        IF finalPosition == 13 THEN
          ;FOLD SPTP P113 Vel=100 % PDAT1 Tool[1]:SMC Base[0] ;%{PE}
          ;FOLD Parameters ;%{h}
          ;Params IlfProvider=kukaroboter.basistech.inlineforms.movement.spline; Kuka.IsGlobalPoint=False; Kuka.PointName=P113; Kuka.BlendingEnabled=False; Kuka.MoveDataPtpName=PDAT1; Kuka.VelocityPtp=100; Kuka.VelocityFieldEnabled=True; Kuka.ColDetectFieldEnabled=True; Kuka.CurrentCDSetIndex=0; Kuka.MovementParameterFieldEnabled=True; IlfCommand=SPTP
          ;ENDFOLD
          SPTP XP113 WITH $VEL_AXIS[1] = SVEL_JOINT(100.0), $TOOL = STOOL2(FP113), $BASE = SBASE(FP113.BASE_NO), $IPO_MODE = SIPO_MODE(FP113.IPO_FRAME), $LOAD = SLOAD(FP113.TOOL_NO), $ACC_AXIS[1] = SACC_JOINT(PPDAT1), $APO = SAPO_PTP(PPDAT1), $GEAR_JERK[1] = SGEAR_JERK(PPDAT1), $COLLMON_TOL_PRO[1] = USE_CM_PRO_VALUES(0)
          ;ENDFOLD
          ;FOLD SLIN P213 Vel=0.1 m/s CPDAT27 Tool[1]:SMC Base[0] ;%{PE}
          ;FOLD Parameters ;%{h}
          ;Params IlfProvider=kukaroboter.basistech.inlineforms.movement.spline; Kuka.IsGlobalPoint=False; Kuka.PointName=P213; Kuka.BlendingEnabled=False; Kuka.MoveDataName=CPDAT27; Kuka.VelocityPath=0.1; Kuka.VelocityFieldEnabled=True; Kuka.ColDetectFieldEnabled=True; Kuka.CurrentCDSetIndex=0; Kuka.MovementParameterFieldEnabled=True; IlfCommand=SLIN
          ;ENDFOLD
          SLIN XP213 WITH $VEL = SVEL_CP(0.1, , LCPDAT27), $TOOL = STOOL2(FP213), $BASE = SBASE(FP213.BASE_NO), $IPO_MODE = SIPO_MODE(FP213.IPO_FRAME), $LOAD = SLOAD(FP213.TOOL_NO), $ACC = SACC_CP(LCPDAT27), $ORI_TYPE = SORI_TYP(LCPDAT27), $APO = SAPO(LCPDAT27), $JERK = SJERK(LCPDAT27), $COLLMON_TOL_PRO[1] = USE_CM_PRO_VALUES(0)
          ;ENDFOLD
          ;FOLD Gripper SET [1]Gripper1 State=[1]ABIERTA Wait 0.2[s] Check with Strategy 1 ;%{PE}
          ;FOLD Parameters Parameters ;%{h}
          ;Params IlfProvider=GripperTech.GripperSet;setgripper=1;setstate=1;setcont=nocont;waittime=0.2;errorstrategy=1
          ;ENDFOLD
          GRPg_SetStateAndCheck(1, 1, 0.2, 1)
          ;ENDFOLD
          ;FOLD SLIN P113 Vel=0.1 m/s CPDAT28 Tool[1]:SMC Base[0] ;%{PE}
          ;FOLD Parameters ;%{h}
          ;Params IlfProvider=kukaroboter.basistech.inlineforms.movement.spline; Kuka.IsGlobalPoint=False; Kuka.PointName=P113; Kuka.BlendingEnabled=False; Kuka.MoveDataName=CPDAT28; Kuka.VelocityPath=0.1; Kuka.VelocityFieldEnabled=True; Kuka.ColDetectFieldEnabled=True; Kuka.CurrentCDSetIndex=0; Kuka.MovementParameterFieldEnabled=True; IlfCommand=SLIN
          ;ENDFOLD
          SLIN XP113 WITH $VEL = SVEL_CP(0.1, , LCPDAT28), $TOOL = STOOL2(FP113), $BASE = SBASE(FP113.BASE_NO), $IPO_MODE = SIPO_MODE(FP113.IPO_FRAME), $LOAD = SLOAD(FP113.TOOL_NO), $ACC = SACC_CP(LCPDAT28), $ORI_TYPE = SORI_TYP(LCPDAT28), $APO = SAPO(LCPDAT28), $JERK = SJERK(LCPDAT28), $COLLMON_TOL_PRO[1] = USE_CM_PRO_VALUES(0)
          ;ENDFOLD
          ;FOLD SPTP P600 Vel=100 % PDAT1 Tool[1]:SMC Base[0] ;%{PE}
          ;FOLD Parameters ;%{h}
          ;Params IlfProvider=kukaroboter.basistech.inlineforms.movement.spline; Kuka.IsGlobalPoint=False; Kuka.PointName=P600; Kuka.BlendingEnabled=False; Kuka.MoveDataPtpName=PDAT1; Kuka.VelocityPtp=100; Kuka.VelocityFieldEnabled=True; Kuka.ColDetectFieldEnabled=True; Kuka.CurrentCDSetIndex=0; Kuka.MovementParameterFieldEnabled=True; IlfCommand=SPTP
          ;ENDFOLD
          SPTP XP600 WITH $VEL_AXIS[1] = SVEL_JOINT(100.0), $TOOL = STOOL2(FP600), $BASE = SBASE(FP600.BASE_NO), $IPO_MODE = SIPO_MODE(FP600.IPO_FRAME), $LOAD = SLOAD(FP600.TOOL_NO), $ACC_AXIS[1] = SACC_JOINT(PPDAT1), $APO = SAPO_PTP(PPDAT1), $GEAR_JERK[1] = SGEAR_JERK(PPDAT1), $COLLMON_TOL_PRO[1] = USE_CM_PRO_VALUES(0)
          ;ENDFOLD
          ;FOLD SLIN P601 Vel=0.1 m/s CPDAT27 Tool[1]:SMC Base[0] ;%{PE}
          ;FOLD Parameters ;%{h}
          ;Params IlfProvider=kukaroboter.basistech.inlineforms.movement.spline; Kuka.IsGlobalPoint=False; Kuka.PointName=P601; Kuka.BlendingEnabled=False; Kuka.MoveDataName=CPDAT27; Kuka.VelocityPath=0.1; Kuka.VelocityFieldEnabled=True; Kuka.ColDetectFieldEnabled=True; Kuka.CurrentCDSetIndex=0; Kuka.MovementParameterFieldEnabled=True; IlfCommand=SLIN
          ;ENDFOLD
          SLIN XP601 WITH $VEL = SVEL_CP(0.1, , LCPDAT27), $TOOL = STOOL2(FP601), $BASE = SBASE(FP601.BASE_NO), $IPO_MODE = SIPO_MODE(FP601.IPO_FRAME), $LOAD = SLOAD(FP601.TOOL_NO), $ACC = SACC_CP(LCPDAT27), $ORI_TYPE = SORI_TYP(LCPDAT27), $APO = SAPO(LCPDAT27), $JERK = SJERK(LCPDAT27), $COLLMON_TOL_PRO[1] = USE_CM_PRO_VALUES(0)
          ;ENDFOLD
          ;FOLD SLIN P602 Vel=0.1 m/s CPDAT27 Tool[1]:SMC Base[0] ;%{PE}
          ;FOLD Parameters ;%{h}
          ;Params IlfProvider=kukaroboter.basistech.inlineforms.movement.spline; Kuka.IsGlobalPoint=False; Kuka.PointName=P602; Kuka.BlendingEnabled=False; Kuka.MoveDataName=CPDAT27; Kuka.VelocityPath=0.1; Kuka.VelocityFieldEnabled=True; Kuka.ColDetectFieldEnabled=True; Kuka.CurrentCDSetIndex=0; Kuka.MovementParameterFieldEnabled=True; IlfCommand=SLIN
          ;ENDFOLD
          SLIN XP602 WITH $VEL = SVEL_CP(0.1, , LCPDAT27), $TOOL = STOOL2(FP602), $BASE = SBASE(FP602.BASE_NO), $IPO_MODE = SIPO_MODE(FP602.IPO_FRAME), $LOAD = SLOAD(FP602.TOOL_NO), $ACC = SACC_CP(LCPDAT27), $ORI_TYPE = SORI_TYP(LCPDAT27), $APO = SAPO(LCPDAT27), $JERK = SJERK(LCPDAT27), $COLLMON_TOL_PRO[1] = USE_CM_PRO_VALUES(0)
          ;ENDFOLD
        ENDIF
        IF finalPosition == 14 THEN
          ;FOLD SPTP P114 Vel=100 % PDAT1 Tool[1]:SMC Base[0] ;%{PE}
          ;FOLD Parameters ;%{h}
          ;Params IlfProvider=kukaroboter.basistech.inlineforms.movement.spline; Kuka.IsGlobalPoint=False; Kuka.PointName=P114; Kuka.BlendingEnabled=False; Kuka.MoveDataPtpName=PDAT1; Kuka.VelocityPtp=100; Kuka.VelocityFieldEnabled=True; Kuka.ColDetectFieldEnabled=True; Kuka.CurrentCDSetIndex=0; Kuka.MovementParameterFieldEnabled=True; IlfCommand=SPTP
          ;ENDFOLD
          SPTP XP114 WITH $VEL_AXIS[1] = SVEL_JOINT(100.0), $TOOL = STOOL2(FP114), $BASE = SBASE(FP114.BASE_NO), $IPO_MODE = SIPO_MODE(FP114.IPO_FRAME), $LOAD = SLOAD(FP114.TOOL_NO), $ACC_AXIS[1] = SACC_JOINT(PPDAT1), $APO = SAPO_PTP(PPDAT1), $GEAR_JERK[1] = SGEAR_JERK(PPDAT1), $COLLMON_TOL_PRO[1] = USE_CM_PRO_VALUES(0)
          ;ENDFOLD
          ;FOLD SLIN P214 Vel=0.1 m/s CPDAT27 Tool[1]:SMC Base[0] ;%{PE}
          ;FOLD Parameters ;%{h}
          ;Params IlfProvider=kukaroboter.basistech.inlineforms.movement.spline; Kuka.IsGlobalPoint=False; Kuka.PointName=P214; Kuka.BlendingEnabled=False; Kuka.MoveDataName=CPDAT27; Kuka.VelocityPath=0.1; Kuka.VelocityFieldEnabled=True; Kuka.ColDetectFieldEnabled=True; Kuka.CurrentCDSetIndex=0; Kuka.MovementParameterFieldEnabled=True; IlfCommand=SLIN
          ;ENDFOLD
          SLIN XP214 WITH $VEL = SVEL_CP(0.1, , LCPDAT27), $TOOL = STOOL2(FP214), $BASE = SBASE(FP214.BASE_NO), $IPO_MODE = SIPO_MODE(FP214.IPO_FRAME), $LOAD = SLOAD(FP214.TOOL_NO), $ACC = SACC_CP(LCPDAT27), $ORI_TYPE = SORI_TYP(LCPDAT27), $APO = SAPO(LCPDAT27), $JERK = SJERK(LCPDAT27), $COLLMON_TOL_PRO[1] = USE_CM_PRO_VALUES(0)
          ;ENDFOLD
          ;FOLD Gripper SET [1]Gripper1 State=[1]ABIERTA Wait 0.2[s] Check with Strategy 1 ;%{PE}
          ;FOLD Parameters Parameters ;%{h}
          ;Params IlfProvider=GripperTech.GripperSet;setgripper=1;setstate=1;setcont=nocont;waittime=0.2;errorstrategy=1
          ;ENDFOLD
          GRPg_SetStateAndCheck(1, 1, 0.2, 1)
          ;ENDFOLD
          ;FOLD SLIN P114 Vel=0.1 m/s CPDAT28 Tool[1]:SMC Base[0] ;%{PE}
          ;FOLD Parameters ;%{h}
          ;Params IlfProvider=kukaroboter.basistech.inlineforms.movement.spline; Kuka.IsGlobalPoint=False; Kuka.PointName=P114; Kuka.BlendingEnabled=False; Kuka.MoveDataName=CPDAT28; Kuka.VelocityPath=0.1; Kuka.VelocityFieldEnabled=True; Kuka.ColDetectFieldEnabled=True; Kuka.CurrentCDSetIndex=0; Kuka.MovementParameterFieldEnabled=True; IlfCommand=SLIN
          ;ENDFOLD
          SLIN XP114 WITH $VEL = SVEL_CP(0.1, , LCPDAT28), $TOOL = STOOL2(FP114), $BASE = SBASE(FP114.BASE_NO), $IPO_MODE = SIPO_MODE(FP114.IPO_FRAME), $LOAD = SLOAD(FP114.TOOL_NO), $ACC = SACC_CP(LCPDAT28), $ORI_TYPE = SORI_TYP(LCPDAT28), $APO = SAPO(LCPDAT28), $JERK = SJERK(LCPDAT28), $COLLMON_TOL_PRO[1] = USE_CM_PRO_VALUES(0)
          ;ENDFOLD
          ;FOLD SPTP P600 Vel=100 % PDAT1 Tool[1]:SMC Base[0] ;%{PE}
          ;FOLD Parameters ;%{h}
          ;Params IlfProvider=kukaroboter.basistech.inlineforms.movement.spline; Kuka.IsGlobalPoint=False; Kuka.PointName=P600; Kuka.BlendingEnabled=False; Kuka.MoveDataPtpName=PDAT1; Kuka.VelocityPtp=100; Kuka.VelocityFieldEnabled=True; Kuka.ColDetectFieldEnabled=True; Kuka.CurrentCDSetIndex=0; Kuka.MovementParameterFieldEnabled=True; IlfCommand=SPTP
          ;ENDFOLD
          SPTP XP600 WITH $VEL_AXIS[1] = SVEL_JOINT(100.0), $TOOL = STOOL2(FP600), $BASE = SBASE(FP600.BASE_NO), $IPO_MODE = SIPO_MODE(FP600.IPO_FRAME), $LOAD = SLOAD(FP600.TOOL_NO), $ACC_AXIS[1] = SACC_JOINT(PPDAT1), $APO = SAPO_PTP(PPDAT1), $GEAR_JERK[1] = SGEAR_JERK(PPDAT1), $COLLMON_TOL_PRO[1] = USE_CM_PRO_VALUES(0)
          ;ENDFOLD
          ;FOLD SLIN P601 Vel=0.1 m/s CPDAT27 Tool[1]:SMC Base[0] ;%{PE}
          ;FOLD Parameters ;%{h}
          ;Params IlfProvider=kukaroboter.basistech.inlineforms.movement.spline; Kuka.IsGlobalPoint=False; Kuka.PointName=P601; Kuka.BlendingEnabled=False; Kuka.MoveDataName=CPDAT27; Kuka.VelocityPath=0.1; Kuka.VelocityFieldEnabled=True; Kuka.ColDetectFieldEnabled=True; Kuka.CurrentCDSetIndex=0; Kuka.MovementParameterFieldEnabled=True; IlfCommand=SLIN
          ;ENDFOLD
          SLIN XP601 WITH $VEL = SVEL_CP(0.1, , LCPDAT27), $TOOL = STOOL2(FP601), $BASE = SBASE(FP601.BASE_NO), $IPO_MODE = SIPO_MODE(FP601.IPO_FRAME), $LOAD = SLOAD(FP601.TOOL_NO), $ACC = SACC_CP(LCPDAT27), $ORI_TYPE = SORI_TYP(LCPDAT27), $APO = SAPO(LCPDAT27), $JERK = SJERK(LCPDAT27), $COLLMON_TOL_PRO[1] = USE_CM_PRO_VALUES(0)
          ;ENDFOLD
          ;FOLD SLIN P602 Vel=0.1 m/s CPDAT27 Tool[1]:SMC Base[0] ;%{PE}
          ;FOLD Parameters ;%{h}
          ;Params IlfProvider=kukaroboter.basistech.inlineforms.movement.spline; Kuka.IsGlobalPoint=False; Kuka.PointName=P602; Kuka.BlendingEnabled=False; Kuka.MoveDataName=CPDAT27; Kuka.VelocityPath=0.1; Kuka.VelocityFieldEnabled=True; Kuka.ColDetectFieldEnabled=True; Kuka.CurrentCDSetIndex=0; Kuka.MovementParameterFieldEnabled=True; IlfCommand=SLIN
          ;ENDFOLD
          SLIN XP602 WITH $VEL = SVEL_CP(0.1, , LCPDAT27), $TOOL = STOOL2(FP602), $BASE = SBASE(FP602.BASE_NO), $IPO_MODE = SIPO_MODE(FP602.IPO_FRAME), $LOAD = SLOAD(FP602.TOOL_NO), $ACC = SACC_CP(LCPDAT27), $ORI_TYPE = SORI_TYP(LCPDAT27), $APO = SAPO(LCPDAT27), $JERK = SJERK(LCPDAT27), $COLLMON_TOL_PRO[1] = USE_CM_PRO_VALUES(0)
          ;ENDFOLD
        ENDIF
        IF finalPosition == 15 THEN
          ;FOLD SPTP P115 Vel=100 % PDAT1 Tool[1]:SMC Base[0] ;%{PE}
          ;FOLD Parameters ;%{h}
          ;Params IlfProvider=kukaroboter.basistech.inlineforms.movement.spline; Kuka.IsGlobalPoint=False; Kuka.PointName=P115; Kuka.BlendingEnabled=False; Kuka.MoveDataPtpName=PDAT1; Kuka.VelocityPtp=100; Kuka.VelocityFieldEnabled=True; Kuka.ColDetectFieldEnabled=True; Kuka.CurrentCDSetIndex=0; Kuka.MovementParameterFieldEnabled=True; IlfCommand=SPTP
          ;ENDFOLD
          SPTP XP115 WITH $VEL_AXIS[1] = SVEL_JOINT(100.0), $TOOL = STOOL2(FP115), $BASE = SBASE(FP115.BASE_NO), $IPO_MODE = SIPO_MODE(FP115.IPO_FRAME), $LOAD = SLOAD(FP115.TOOL_NO), $ACC_AXIS[1] = SACC_JOINT(PPDAT1), $APO = SAPO_PTP(PPDAT1), $GEAR_JERK[1] = SGEAR_JERK(PPDAT1), $COLLMON_TOL_PRO[1] = USE_CM_PRO_VALUES(0)
          ;ENDFOLD
          ;FOLD SLIN P215 Vel=0.1 m/s CPDAT27 Tool[1]:SMC Base[0] ;%{PE}
          ;FOLD Parameters ;%{h}
          ;Params IlfProvider=kukaroboter.basistech.inlineforms.movement.spline; Kuka.IsGlobalPoint=False; Kuka.PointName=P215; Kuka.BlendingEnabled=False; Kuka.MoveDataName=CPDAT27; Kuka.VelocityPath=0.1; Kuka.VelocityFieldEnabled=True; Kuka.ColDetectFieldEnabled=True; Kuka.CurrentCDSetIndex=0; Kuka.MovementParameterFieldEnabled=True; IlfCommand=SLIN
          ;ENDFOLD
          SLIN XP215 WITH $VEL = SVEL_CP(0.1, , LCPDAT27), $TOOL = STOOL2(FP215), $BASE = SBASE(FP215.BASE_NO), $IPO_MODE = SIPO_MODE(FP215.IPO_FRAME), $LOAD = SLOAD(FP215.TOOL_NO), $ACC = SACC_CP(LCPDAT27), $ORI_TYPE = SORI_TYP(LCPDAT27), $APO = SAPO(LCPDAT27), $JERK = SJERK(LCPDAT27), $COLLMON_TOL_PRO[1] = USE_CM_PRO_VALUES(0)
          ;ENDFOLD
          ;FOLD Gripper SET [1]Gripper1 State=[1]ABIERTA Wait 0.2[s] Check with Strategy 1 ;%{PE}
          ;FOLD Parameters Parameters ;%{h}
          ;Params IlfProvider=GripperTech.GripperSet;setgripper=1;setstate=1;setcont=nocont;waittime=0.2;errorstrategy=1
          ;ENDFOLD
          GRPg_SetStateAndCheck(1, 1, 0.2, 1)
          ;ENDFOLD
          ;FOLD SLIN P115 Vel=0.1 m/s CPDAT28 Tool[1]:SMC Base[0] ;%{PE}
          ;FOLD Parameters ;%{h}
          ;Params IlfProvider=kukaroboter.basistech.inlineforms.movement.spline; Kuka.IsGlobalPoint=False; Kuka.PointName=P115; Kuka.BlendingEnabled=False; Kuka.MoveDataName=CPDAT28; Kuka.VelocityPath=0.1; Kuka.VelocityFieldEnabled=True; Kuka.ColDetectFieldEnabled=True; Kuka.CurrentCDSetIndex=0; Kuka.MovementParameterFieldEnabled=True; IlfCommand=SLIN
          ;ENDFOLD
          SLIN XP115 WITH $VEL = SVEL_CP(0.1, , LCPDAT28), $TOOL = STOOL2(FP115), $BASE = SBASE(FP115.BASE_NO), $IPO_MODE = SIPO_MODE(FP115.IPO_FRAME), $LOAD = SLOAD(FP115.TOOL_NO), $ACC = SACC_CP(LCPDAT28), $ORI_TYPE = SORI_TYP(LCPDAT28), $APO = SAPO(LCPDAT28), $JERK = SJERK(LCPDAT28), $COLLMON_TOL_PRO[1] = USE_CM_PRO_VALUES(0)
          ;ENDFOLD
          ;FOLD SPTP P600 Vel=100 % PDAT1 Tool[1]:SMC Base[0] ;%{PE}
          ;FOLD Parameters ;%{h}
          ;Params IlfProvider=kukaroboter.basistech.inlineforms.movement.spline; Kuka.IsGlobalPoint=False; Kuka.PointName=P600; Kuka.BlendingEnabled=False; Kuka.MoveDataPtpName=PDAT1; Kuka.VelocityPtp=100; Kuka.VelocityFieldEnabled=True; Kuka.ColDetectFieldEnabled=True; Kuka.CurrentCDSetIndex=0; Kuka.MovementParameterFieldEnabled=True; IlfCommand=SPTP
          ;ENDFOLD
          SPTP XP600 WITH $VEL_AXIS[1] = SVEL_JOINT(100.0), $TOOL = STOOL2(FP600), $BASE = SBASE(FP600.BASE_NO), $IPO_MODE = SIPO_MODE(FP600.IPO_FRAME), $LOAD = SLOAD(FP600.TOOL_NO), $ACC_AXIS[1] = SACC_JOINT(PPDAT1), $APO = SAPO_PTP(PPDAT1), $GEAR_JERK[1] = SGEAR_JERK(PPDAT1), $COLLMON_TOL_PRO[1] = USE_CM_PRO_VALUES(0)
          ;ENDFOLD
          ;FOLD SLIN P601 Vel=0.1 m/s CPDAT27 Tool[1]:SMC Base[0] ;%{PE}
          ;FOLD Parameters ;%{h}
          ;Params IlfProvider=kukaroboter.basistech.inlineforms.movement.spline; Kuka.IsGlobalPoint=False; Kuka.PointName=P601; Kuka.BlendingEnabled=False; Kuka.MoveDataName=CPDAT27; Kuka.VelocityPath=0.1; Kuka.VelocityFieldEnabled=True; Kuka.ColDetectFieldEnabled=True; Kuka.CurrentCDSetIndex=0; Kuka.MovementParameterFieldEnabled=True; IlfCommand=SLIN
          ;ENDFOLD
          SLIN XP601 WITH $VEL = SVEL_CP(0.1, , LCPDAT27), $TOOL = STOOL2(FP601), $BASE = SBASE(FP601.BASE_NO), $IPO_MODE = SIPO_MODE(FP601.IPO_FRAME), $LOAD = SLOAD(FP601.TOOL_NO), $ACC = SACC_CP(LCPDAT27), $ORI_TYPE = SORI_TYP(LCPDAT27), $APO = SAPO(LCPDAT27), $JERK = SJERK(LCPDAT27), $COLLMON_TOL_PRO[1] = USE_CM_PRO_VALUES(0)
          ;ENDFOLD
          ;FOLD SLIN P602 Vel=0.1 m/s CPDAT27 Tool[1]:SMC Base[0] ;%{PE}
          ;FOLD Parameters ;%{h}
          ;Params IlfProvider=kukaroboter.basistech.inlineforms.movement.spline; Kuka.IsGlobalPoint=False; Kuka.PointName=P602; Kuka.BlendingEnabled=False; Kuka.MoveDataName=CPDAT27; Kuka.VelocityPath=0.1; Kuka.VelocityFieldEnabled=True; Kuka.ColDetectFieldEnabled=True; Kuka.CurrentCDSetIndex=0; Kuka.MovementParameterFieldEnabled=True; IlfCommand=SLIN
          ;ENDFOLD
          SLIN XP602 WITH $VEL = SVEL_CP(0.1, , LCPDAT27), $TOOL = STOOL2(FP602), $BASE = SBASE(FP602.BASE_NO), $IPO_MODE = SIPO_MODE(FP602.IPO_FRAME), $LOAD = SLOAD(FP602.TOOL_NO), $ACC = SACC_CP(LCPDAT27), $ORI_TYPE = SORI_TYP(LCPDAT27), $APO = SAPO(LCPDAT27), $JERK = SJERK(LCPDAT27), $COLLMON_TOL_PRO[1] = USE_CM_PRO_VALUES(0)
          ;ENDFOLD
        ENDIF
        IF finalPosition == 16 THEN
          ;FOLD SPTP P116 Vel=100 % PDAT1 Tool[1]:SMC Base[0] ;%{PE}
          ;FOLD Parameters ;%{h}
          ;Params IlfProvider=kukaroboter.basistech.inlineforms.movement.spline; Kuka.IsGlobalPoint=False; Kuka.PointName=P116; Kuka.BlendingEnabled=False; Kuka.MoveDataPtpName=PDAT1; Kuka.VelocityPtp=100; Kuka.VelocityFieldEnabled=True; Kuka.ColDetectFieldEnabled=True; Kuka.CurrentCDSetIndex=0; Kuka.MovementParameterFieldEnabled=True; IlfCommand=SPTP
          ;ENDFOLD
          SPTP XP116 WITH $VEL_AXIS[1] = SVEL_JOINT(100.0), $TOOL = STOOL2(FP116), $BASE = SBASE(FP116.BASE_NO), $IPO_MODE = SIPO_MODE(FP116.IPO_FRAME), $LOAD = SLOAD(FP116.TOOL_NO), $ACC_AXIS[1] = SACC_JOINT(PPDAT1), $APO = SAPO_PTP(PPDAT1), $GEAR_JERK[1] = SGEAR_JERK(PPDAT1), $COLLMON_TOL_PRO[1] = USE_CM_PRO_VALUES(0)
          ;ENDFOLD
          ;FOLD SLIN P216 Vel=0.1 m/s CPDAT27 Tool[1]:SMC Base[0] ;%{PE}
          ;FOLD Parameters ;%{h}
          ;Params IlfProvider=kukaroboter.basistech.inlineforms.movement.spline; Kuka.IsGlobalPoint=False; Kuka.PointName=P216; Kuka.BlendingEnabled=False; Kuka.MoveDataName=CPDAT27; Kuka.VelocityPath=0.1; Kuka.VelocityFieldEnabled=True; Kuka.ColDetectFieldEnabled=True; Kuka.CurrentCDSetIndex=0; Kuka.MovementParameterFieldEnabled=True; IlfCommand=SLIN
          ;ENDFOLD
          SLIN XP216 WITH $VEL = SVEL_CP(0.1, , LCPDAT27), $TOOL = STOOL2(FP216), $BASE = SBASE(FP216.BASE_NO), $IPO_MODE = SIPO_MODE(FP216.IPO_FRAME), $LOAD = SLOAD(FP216.TOOL_NO), $ACC = SACC_CP(LCPDAT27), $ORI_TYPE = SORI_TYP(LCPDAT27), $APO = SAPO(LCPDAT27), $JERK = SJERK(LCPDAT27), $COLLMON_TOL_PRO[1] = USE_CM_PRO_VALUES(0)
          ;ENDFOLD
          ;FOLD Gripper SET [1]Gripper1 State=[1]ABIERTA Wait 0.2[s] Check with Strategy 1 ;%{PE}
          ;FOLD Parameters Parameters ;%{h}
          ;Params IlfProvider=GripperTech.GripperSet;setgripper=1;setstate=1;setcont=nocont;waittime=0.2;errorstrategy=1
          ;ENDFOLD
          GRPg_SetStateAndCheck(1, 1, 0.2, 1)
          ;ENDFOLD
          ;FOLD SLIN P116 Vel=0.1 m/s CPDAT28 Tool[1]:SMC Base[0] ;%{PE}
          ;FOLD Parameters ;%{h}
          ;Params IlfProvider=kukaroboter.basistech.inlineforms.movement.spline; Kuka.IsGlobalPoint=False; Kuka.PointName=P116; Kuka.BlendingEnabled=False; Kuka.MoveDataName=CPDAT28; Kuka.VelocityPath=0.1; Kuka.VelocityFieldEnabled=True; Kuka.ColDetectFieldEnabled=True; Kuka.CurrentCDSetIndex=0; Kuka.MovementParameterFieldEnabled=True; IlfCommand=SLIN
          ;ENDFOLD
          SLIN XP116 WITH $VEL = SVEL_CP(0.1, , LCPDAT28), $TOOL = STOOL2(FP116), $BASE = SBASE(FP116.BASE_NO), $IPO_MODE = SIPO_MODE(FP116.IPO_FRAME), $LOAD = SLOAD(FP116.TOOL_NO), $ACC = SACC_CP(LCPDAT28), $ORI_TYPE = SORI_TYP(LCPDAT28), $APO = SAPO(LCPDAT28), $JERK = SJERK(LCPDAT28), $COLLMON_TOL_PRO[1] = USE_CM_PRO_VALUES(0)
          ;ENDFOLD
          ;FOLD SPTP P600 Vel=100 % PDAT1 Tool[1]:SMC Base[0] ;%{PE}
          ;FOLD Parameters ;%{h}
          ;Params IlfProvider=kukaroboter.basistech.inlineforms.movement.spline; Kuka.IsGlobalPoint=False; Kuka.PointName=P600; Kuka.BlendingEnabled=False; Kuka.MoveDataPtpName=PDAT1; Kuka.VelocityPtp=100; Kuka.VelocityFieldEnabled=True; Kuka.ColDetectFieldEnabled=True; Kuka.CurrentCDSetIndex=0; Kuka.MovementParameterFieldEnabled=True; IlfCommand=SPTP
          ;ENDFOLD
          SPTP XP600 WITH $VEL_AXIS[1] = SVEL_JOINT(100.0), $TOOL = STOOL2(FP600), $BASE = SBASE(FP600.BASE_NO), $IPO_MODE = SIPO_MODE(FP600.IPO_FRAME), $LOAD = SLOAD(FP600.TOOL_NO), $ACC_AXIS[1] = SACC_JOINT(PPDAT1), $APO = SAPO_PTP(PPDAT1), $GEAR_JERK[1] = SGEAR_JERK(PPDAT1), $COLLMON_TOL_PRO[1] = USE_CM_PRO_VALUES(0)
          ;ENDFOLD
          ;FOLD SLIN P601 Vel=0.1 m/s CPDAT27 Tool[1]:SMC Base[0] ;%{PE}
          ;FOLD Parameters ;%{h}
          ;Params IlfProvider=kukaroboter.basistech.inlineforms.movement.spline; Kuka.IsGlobalPoint=False; Kuka.PointName=P601; Kuka.BlendingEnabled=False; Kuka.MoveDataName=CPDAT27; Kuka.VelocityPath=0.1; Kuka.VelocityFieldEnabled=True; Kuka.ColDetectFieldEnabled=True; Kuka.CurrentCDSetIndex=0; Kuka.MovementParameterFieldEnabled=True; IlfCommand=SLIN
          ;ENDFOLD
          SLIN XP601 WITH $VEL = SVEL_CP(0.1, , LCPDAT27), $TOOL = STOOL2(FP601), $BASE = SBASE(FP601.BASE_NO), $IPO_MODE = SIPO_MODE(FP601.IPO_FRAME), $LOAD = SLOAD(FP601.TOOL_NO), $ACC = SACC_CP(LCPDAT27), $ORI_TYPE = SORI_TYP(LCPDAT27), $APO = SAPO(LCPDAT27), $JERK = SJERK(LCPDAT27), $COLLMON_TOL_PRO[1] = USE_CM_PRO_VALUES(0)
          ;ENDFOLD
          ;FOLD SLIN P602 Vel=0.1 m/s CPDAT27 Tool[1]:SMC Base[0] ;%{PE}
          ;FOLD Parameters ;%{h}
          ;Params IlfProvider=kukaroboter.basistech.inlineforms.movement.spline; Kuka.IsGlobalPoint=False; Kuka.PointName=P602; Kuka.BlendingEnabled=False; Kuka.MoveDataName=CPDAT27; Kuka.VelocityPath=0.1; Kuka.VelocityFieldEnabled=True; Kuka.ColDetectFieldEnabled=True; Kuka.CurrentCDSetIndex=0; Kuka.MovementParameterFieldEnabled=True; IlfCommand=SLIN
          ;ENDFOLD
          SLIN XP602 WITH $VEL = SVEL_CP(0.1, , LCPDAT27), $TOOL = STOOL2(FP602), $BASE = SBASE(FP602.BASE_NO), $IPO_MODE = SIPO_MODE(FP602.IPO_FRAME), $LOAD = SLOAD(FP602.TOOL_NO), $ACC = SACC_CP(LCPDAT27), $ORI_TYPE = SORI_TYP(LCPDAT27), $APO = SAPO(LCPDAT27), $JERK = SJERK(LCPDAT27), $COLLMON_TOL_PRO[1] = USE_CM_PRO_VALUES(0)
          ;ENDFOLD
        ENDIF
        IF finalPosition == 17 THEN
          ;FOLD SPTP P117 Vel=100 % PDAT1 Tool[1]:SMC Base[0] ;%{PE}
          ;FOLD Parameters ;%{h}
          ;Params IlfProvider=kukaroboter.basistech.inlineforms.movement.spline; Kuka.IsGlobalPoint=False; Kuka.PointName=P117; Kuka.BlendingEnabled=False; Kuka.MoveDataPtpName=PDAT1; Kuka.VelocityPtp=100; Kuka.VelocityFieldEnabled=True; Kuka.ColDetectFieldEnabled=True; Kuka.CurrentCDSetIndex=0; Kuka.MovementParameterFieldEnabled=True; IlfCommand=SPTP
          ;ENDFOLD
          SPTP XP117 WITH $VEL_AXIS[1] = SVEL_JOINT(100.0), $TOOL = STOOL2(FP117), $BASE = SBASE(FP117.BASE_NO), $IPO_MODE = SIPO_MODE(FP117.IPO_FRAME), $LOAD = SLOAD(FP117.TOOL_NO), $ACC_AXIS[1] = SACC_JOINT(PPDAT1), $APO = SAPO_PTP(PPDAT1), $GEAR_JERK[1] = SGEAR_JERK(PPDAT1), $COLLMON_TOL_PRO[1] = USE_CM_PRO_VALUES(0)
          ;ENDFOLD
          ;FOLD SLIN P217 Vel=0.1 m/s CPDAT27 Tool[1]:SMC Base[0] ;%{PE}
          ;FOLD Parameters ;%{h}
          ;Params IlfProvider=kukaroboter.basistech.inlineforms.movement.spline; Kuka.IsGlobalPoint=False; Kuka.PointName=P217; Kuka.BlendingEnabled=False; Kuka.MoveDataName=CPDAT27; Kuka.VelocityPath=0.1; Kuka.VelocityFieldEnabled=True; Kuka.ColDetectFieldEnabled=True; Kuka.CurrentCDSetIndex=0; Kuka.MovementParameterFieldEnabled=True; IlfCommand=SLIN
          ;ENDFOLD
          SLIN XP217 WITH $VEL = SVEL_CP(0.1, , LCPDAT27), $TOOL = STOOL2(FP217), $BASE = SBASE(FP217.BASE_NO), $IPO_MODE = SIPO_MODE(FP217.IPO_FRAME), $LOAD = SLOAD(FP217.TOOL_NO), $ACC = SACC_CP(LCPDAT27), $ORI_TYPE = SORI_TYP(LCPDAT27), $APO = SAPO(LCPDAT27), $JERK = SJERK(LCPDAT27), $COLLMON_TOL_PRO[1] = USE_CM_PRO_VALUES(0)
          ;ENDFOLD
          ;FOLD Gripper SET [1]Gripper1 State=[1]ABIERTA Wait 0.2[s] Check with Strategy 1 ;%{PE}
          ;FOLD Parameters Parameters ;%{h}
          ;Params IlfProvider=GripperTech.GripperSet;setgripper=1;setstate=1;setcont=nocont;waittime=0.2;errorstrategy=1
          ;ENDFOLD
          GRPg_SetStateAndCheck(1, 1, 0.2, 1)
          ;ENDFOLD
          ;FOLD SLIN P117 Vel=0.1 m/s CPDAT28 Tool[1]:SMC Base[0] ;%{PE}
          ;FOLD Parameters ;%{h}
          ;Params IlfProvider=kukaroboter.basistech.inlineforms.movement.spline; Kuka.IsGlobalPoint=False; Kuka.PointName=P117; Kuka.BlendingEnabled=False; Kuka.MoveDataName=CPDAT28; Kuka.VelocityPath=0.1; Kuka.VelocityFieldEnabled=True; Kuka.ColDetectFieldEnabled=True; Kuka.CurrentCDSetIndex=0; Kuka.MovementParameterFieldEnabled=True; IlfCommand=SLIN
          ;ENDFOLD
          SLIN XP117 WITH $VEL = SVEL_CP(0.1, , LCPDAT28), $TOOL = STOOL2(FP117), $BASE = SBASE(FP117.BASE_NO), $IPO_MODE = SIPO_MODE(FP117.IPO_FRAME), $LOAD = SLOAD(FP117.TOOL_NO), $ACC = SACC_CP(LCPDAT28), $ORI_TYPE = SORI_TYP(LCPDAT28), $APO = SAPO(LCPDAT28), $JERK = SJERK(LCPDAT28), $COLLMON_TOL_PRO[1] = USE_CM_PRO_VALUES(0)
          ;ENDFOLD
          ;FOLD SPTP P600 Vel=100 % PDAT1 Tool[1]:SMC Base[0] ;%{PE}
          ;FOLD Parameters ;%{h}
          ;Params IlfProvider=kukaroboter.basistech.inlineforms.movement.spline; Kuka.IsGlobalPoint=False; Kuka.PointName=P600; Kuka.BlendingEnabled=False; Kuka.MoveDataPtpName=PDAT1; Kuka.VelocityPtp=100; Kuka.VelocityFieldEnabled=True; Kuka.ColDetectFieldEnabled=True; Kuka.CurrentCDSetIndex=0; Kuka.MovementParameterFieldEnabled=True; IlfCommand=SPTP
          ;ENDFOLD
          SPTP XP600 WITH $VEL_AXIS[1] = SVEL_JOINT(100.0), $TOOL = STOOL2(FP600), $BASE = SBASE(FP600.BASE_NO), $IPO_MODE = SIPO_MODE(FP600.IPO_FRAME), $LOAD = SLOAD(FP600.TOOL_NO), $ACC_AXIS[1] = SACC_JOINT(PPDAT1), $APO = SAPO_PTP(PPDAT1), $GEAR_JERK[1] = SGEAR_JERK(PPDAT1), $COLLMON_TOL_PRO[1] = USE_CM_PRO_VALUES(0)
          ;ENDFOLD
          ;FOLD SLIN P601 Vel=0.1 m/s CPDAT27 Tool[1]:SMC Base[0] ;%{PE}
          ;FOLD Parameters ;%{h}
          ;Params IlfProvider=kukaroboter.basistech.inlineforms.movement.spline; Kuka.IsGlobalPoint=False; Kuka.PointName=P601; Kuka.BlendingEnabled=False; Kuka.MoveDataName=CPDAT27; Kuka.VelocityPath=0.1; Kuka.VelocityFieldEnabled=True; Kuka.ColDetectFieldEnabled=True; Kuka.CurrentCDSetIndex=0; Kuka.MovementParameterFieldEnabled=True; IlfCommand=SLIN
          ;ENDFOLD
          SLIN XP601 WITH $VEL = SVEL_CP(0.1, , LCPDAT27), $TOOL = STOOL2(FP601), $BASE = SBASE(FP601.BASE_NO), $IPO_MODE = SIPO_MODE(FP601.IPO_FRAME), $LOAD = SLOAD(FP601.TOOL_NO), $ACC = SACC_CP(LCPDAT27), $ORI_TYPE = SORI_TYP(LCPDAT27), $APO = SAPO(LCPDAT27), $JERK = SJERK(LCPDAT27), $COLLMON_TOL_PRO[1] = USE_CM_PRO_VALUES(0)
          ;ENDFOLD
          ;FOLD SLIN P602 Vel=0.1 m/s CPDAT27 Tool[1]:SMC Base[0] ;%{PE}
          ;FOLD Parameters ;%{h}
          ;Params IlfProvider=kukaroboter.basistech.inlineforms.movement.spline; Kuka.IsGlobalPoint=False; Kuka.PointName=P602; Kuka.BlendingEnabled=False; Kuka.MoveDataName=CPDAT27; Kuka.VelocityPath=0.1; Kuka.VelocityFieldEnabled=True; Kuka.ColDetectFieldEnabled=True; Kuka.CurrentCDSetIndex=0; Kuka.MovementParameterFieldEnabled=True; IlfCommand=SLIN
          ;ENDFOLD
          SLIN XP602 WITH $VEL = SVEL_CP(0.1, , LCPDAT27), $TOOL = STOOL2(FP602), $BASE = SBASE(FP602.BASE_NO), $IPO_MODE = SIPO_MODE(FP602.IPO_FRAME), $LOAD = SLOAD(FP602.TOOL_NO), $ACC = SACC_CP(LCPDAT27), $ORI_TYPE = SORI_TYP(LCPDAT27), $APO = SAPO(LCPDAT27), $JERK = SJERK(LCPDAT27), $COLLMON_TOL_PRO[1] = USE_CM_PRO_VALUES(0)
          ;ENDFOLD
        ENDIF
        IF finalPosition == 18 THEN
          ;FOLD SPTP P118 Vel=100 % PDAT1 Tool[1]:SMC Base[0] ;%{PE}
          ;FOLD Parameters ;%{h}
          ;Params IlfProvider=kukaroboter.basistech.inlineforms.movement.spline; Kuka.IsGlobalPoint=False; Kuka.PointName=P118; Kuka.BlendingEnabled=False; Kuka.MoveDataPtpName=PDAT1; Kuka.VelocityPtp=100; Kuka.VelocityFieldEnabled=True; Kuka.ColDetectFieldEnabled=True; Kuka.CurrentCDSetIndex=0; Kuka.MovementParameterFieldEnabled=True; IlfCommand=SPTP
          ;ENDFOLD
          SPTP XP118 WITH $VEL_AXIS[1] = SVEL_JOINT(100.0), $TOOL = STOOL2(FP118), $BASE = SBASE(FP118.BASE_NO), $IPO_MODE = SIPO_MODE(FP118.IPO_FRAME), $LOAD = SLOAD(FP118.TOOL_NO), $ACC_AXIS[1] = SACC_JOINT(PPDAT1), $APO = SAPO_PTP(PPDAT1), $GEAR_JERK[1] = SGEAR_JERK(PPDAT1), $COLLMON_TOL_PRO[1] = USE_CM_PRO_VALUES(0)
          ;ENDFOLD
          ;FOLD SLIN P218 Vel=0.1 m/s CPDAT27 Tool[1]:SMC Base[0] ;%{PE}
          ;FOLD Parameters ;%{h}
          ;Params IlfProvider=kukaroboter.basistech.inlineforms.movement.spline; Kuka.IsGlobalPoint=False; Kuka.PointName=P218; Kuka.BlendingEnabled=False; Kuka.MoveDataName=CPDAT27; Kuka.VelocityPath=0.1; Kuka.VelocityFieldEnabled=True; Kuka.ColDetectFieldEnabled=True; Kuka.CurrentCDSetIndex=0; Kuka.MovementParameterFieldEnabled=True; IlfCommand=SLIN
          ;ENDFOLD
          SLIN XP218 WITH $VEL = SVEL_CP(0.1, , LCPDAT27), $TOOL = STOOL2(FP218), $BASE = SBASE(FP218.BASE_NO), $IPO_MODE = SIPO_MODE(FP218.IPO_FRAME), $LOAD = SLOAD(FP218.TOOL_NO), $ACC = SACC_CP(LCPDAT27), $ORI_TYPE = SORI_TYP(LCPDAT27), $APO = SAPO(LCPDAT27), $JERK = SJERK(LCPDAT27), $COLLMON_TOL_PRO[1] = USE_CM_PRO_VALUES(0)
          ;ENDFOLD
          ;FOLD Gripper SET [1]Gripper1 State=[1]ABIERTA Wait 0.2[s] Check with Strategy 1 ;%{PE}
          ;FOLD Parameters Parameters ;%{h}
          ;Params IlfProvider=GripperTech.GripperSet;setgripper=1;setstate=1;setcont=nocont;waittime=0.2;errorstrategy=1
          ;ENDFOLD
          GRPg_SetStateAndCheck(1, 1, 0.2, 1)
          ;ENDFOLD
          ;FOLD SLIN P118 Vel=0.1 m/s CPDAT28 Tool[1]:SMC Base[0] ;%{PE}
          ;FOLD Parameters ;%{h}
          ;Params IlfProvider=kukaroboter.basistech.inlineforms.movement.spline; Kuka.IsGlobalPoint=False; Kuka.PointName=P118; Kuka.BlendingEnabled=False; Kuka.MoveDataName=CPDAT28; Kuka.VelocityPath=0.1; Kuka.VelocityFieldEnabled=True; Kuka.ColDetectFieldEnabled=True; Kuka.CurrentCDSetIndex=0; Kuka.MovementParameterFieldEnabled=True; IlfCommand=SLIN
          ;ENDFOLD
          SLIN XP118 WITH $VEL = SVEL_CP(0.1, , LCPDAT28), $TOOL = STOOL2(FP118), $BASE = SBASE(FP118.BASE_NO), $IPO_MODE = SIPO_MODE(FP118.IPO_FRAME), $LOAD = SLOAD(FP118.TOOL_NO), $ACC = SACC_CP(LCPDAT28), $ORI_TYPE = SORI_TYP(LCPDAT28), $APO = SAPO(LCPDAT28), $JERK = SJERK(LCPDAT28), $COLLMON_TOL_PRO[1] = USE_CM_PRO_VALUES(0)
          ;ENDFOLD
          ;FOLD SPTP P600 Vel=100 % PDAT1 Tool[1]:SMC Base[0] ;%{PE}
          ;FOLD Parameters ;%{h}
          ;Params IlfProvider=kukaroboter.basistech.inlineforms.movement.spline; Kuka.IsGlobalPoint=False; Kuka.PointName=P600; Kuka.BlendingEnabled=False; Kuka.MoveDataPtpName=PDAT1; Kuka.VelocityPtp=100; Kuka.VelocityFieldEnabled=True; Kuka.ColDetectFieldEnabled=True; Kuka.CurrentCDSetIndex=0; Kuka.MovementParameterFieldEnabled=True; IlfCommand=SPTP
          ;ENDFOLD
          SPTP XP600 WITH $VEL_AXIS[1] = SVEL_JOINT(100.0), $TOOL = STOOL2(FP600), $BASE = SBASE(FP600.BASE_NO), $IPO_MODE = SIPO_MODE(FP600.IPO_FRAME), $LOAD = SLOAD(FP600.TOOL_NO), $ACC_AXIS[1] = SACC_JOINT(PPDAT1), $APO = SAPO_PTP(PPDAT1), $GEAR_JERK[1] = SGEAR_JERK(PPDAT1), $COLLMON_TOL_PRO[1] = USE_CM_PRO_VALUES(0)
          ;ENDFOLD
          ;FOLD SLIN P601 Vel=0.1 m/s CPDAT27 Tool[1]:SMC Base[0] ;%{PE}
          ;FOLD Parameters ;%{h}
          ;Params IlfProvider=kukaroboter.basistech.inlineforms.movement.spline; Kuka.IsGlobalPoint=False; Kuka.PointName=P601; Kuka.BlendingEnabled=False; Kuka.MoveDataName=CPDAT27; Kuka.VelocityPath=0.1; Kuka.VelocityFieldEnabled=True; Kuka.ColDetectFieldEnabled=True; Kuka.CurrentCDSetIndex=0; Kuka.MovementParameterFieldEnabled=True; IlfCommand=SLIN
          ;ENDFOLD
          SLIN XP601 WITH $VEL = SVEL_CP(0.1, , LCPDAT27), $TOOL = STOOL2(FP601), $BASE = SBASE(FP601.BASE_NO), $IPO_MODE = SIPO_MODE(FP601.IPO_FRAME), $LOAD = SLOAD(FP601.TOOL_NO), $ACC = SACC_CP(LCPDAT27), $ORI_TYPE = SORI_TYP(LCPDAT27), $APO = SAPO(LCPDAT27), $JERK = SJERK(LCPDAT27), $COLLMON_TOL_PRO[1] = USE_CM_PRO_VALUES(0)
          ;ENDFOLD
          ;FOLD SLIN P602 Vel=0.1 m/s CPDAT27 Tool[1]:SMC Base[0] ;%{PE}
          ;FOLD Parameters ;%{h}
          ;Params IlfProvider=kukaroboter.basistech.inlineforms.movement.spline; Kuka.IsGlobalPoint=False; Kuka.PointName=P602; Kuka.BlendingEnabled=False; Kuka.MoveDataName=CPDAT27; Kuka.VelocityPath=0.1; Kuka.VelocityFieldEnabled=True; Kuka.ColDetectFieldEnabled=True; Kuka.CurrentCDSetIndex=0; Kuka.MovementParameterFieldEnabled=True; IlfCommand=SLIN
          ;ENDFOLD
          SLIN XP602 WITH $VEL = SVEL_CP(0.1, , LCPDAT27), $TOOL = STOOL2(FP602), $BASE = SBASE(FP602.BASE_NO), $IPO_MODE = SIPO_MODE(FP602.IPO_FRAME), $LOAD = SLOAD(FP602.TOOL_NO), $ACC = SACC_CP(LCPDAT27), $ORI_TYPE = SORI_TYP(LCPDAT27), $APO = SAPO(LCPDAT27), $JERK = SJERK(LCPDAT27), $COLLMON_TOL_PRO[1] = USE_CM_PRO_VALUES(0)
          ;ENDFOLD
        ENDIF
        IF finalPosition == 19 THEN
          ;FOLD SPTP P119 Vel=100 % PDAT1 Tool[1]:SMC Base[0] ;%{PE}
          ;FOLD Parameters ;%{h}
          ;Params IlfProvider=kukaroboter.basistech.inlineforms.movement.spline; Kuka.IsGlobalPoint=False; Kuka.PointName=P119; Kuka.BlendingEnabled=False; Kuka.MoveDataPtpName=PDAT1; Kuka.VelocityPtp=100; Kuka.VelocityFieldEnabled=True; Kuka.ColDetectFieldEnabled=True; Kuka.CurrentCDSetIndex=0; Kuka.MovementParameterFieldEnabled=True; IlfCommand=SPTP
          ;ENDFOLD
          SPTP XP119 WITH $VEL_AXIS[1] = SVEL_JOINT(100.0), $TOOL = STOOL2(FP119), $BASE = SBASE(FP119.BASE_NO), $IPO_MODE = SIPO_MODE(FP119.IPO_FRAME), $LOAD = SLOAD(FP119.TOOL_NO), $ACC_AXIS[1] = SACC_JOINT(PPDAT1), $APO = SAPO_PTP(PPDAT1), $GEAR_JERK[1] = SGEAR_JERK(PPDAT1), $COLLMON_TOL_PRO[1] = USE_CM_PRO_VALUES(0)
          ;ENDFOLD
          ;FOLD SLIN P219 Vel=0.1 m/s CPDAT27 Tool[1]:SMC Base[0] ;%{PE}
          ;FOLD Parameters ;%{h}
          ;Params IlfProvider=kukaroboter.basistech.inlineforms.movement.spline; Kuka.IsGlobalPoint=False; Kuka.PointName=P219; Kuka.BlendingEnabled=False; Kuka.MoveDataName=CPDAT27; Kuka.VelocityPath=0.1; Kuka.VelocityFieldEnabled=True; Kuka.ColDetectFieldEnabled=True; Kuka.CurrentCDSetIndex=0; Kuka.MovementParameterFieldEnabled=True; IlfCommand=SLIN
          ;ENDFOLD
          SLIN XP219 WITH $VEL = SVEL_CP(0.1, , LCPDAT27), $TOOL = STOOL2(FP219), $BASE = SBASE(FP219.BASE_NO), $IPO_MODE = SIPO_MODE(FP219.IPO_FRAME), $LOAD = SLOAD(FP219.TOOL_NO), $ACC = SACC_CP(LCPDAT27), $ORI_TYPE = SORI_TYP(LCPDAT27), $APO = SAPO(LCPDAT27), $JERK = SJERK(LCPDAT27), $COLLMON_TOL_PRO[1] = USE_CM_PRO_VALUES(0)
          ;ENDFOLD
          ;FOLD Gripper SET [1]Gripper1 State=[1]ABIERTA Wait 0.2[s] Check with Strategy 1 ;%{PE}
          ;FOLD Parameters Parameters ;%{h}
          ;Params IlfProvider=GripperTech.GripperSet;setgripper=1;setstate=1;setcont=nocont;waittime=0.2;errorstrategy=1
          ;ENDFOLD
          GRPg_SetStateAndCheck(1, 1, 0.2, 1)
          ;ENDFOLD
          ;FOLD SLIN P119 Vel=0.1 m/s CPDAT28 Tool[1]:SMC Base[0] ;%{PE}
          ;FOLD Parameters ;%{h}
          ;Params IlfProvider=kukaroboter.basistech.inlineforms.movement.spline; Kuka.IsGlobalPoint=False; Kuka.PointName=P119; Kuka.BlendingEnabled=False; Kuka.MoveDataName=CPDAT28; Kuka.VelocityPath=0.1; Kuka.VelocityFieldEnabled=True; Kuka.ColDetectFieldEnabled=True; Kuka.CurrentCDSetIndex=0; Kuka.MovementParameterFieldEnabled=True; IlfCommand=SLIN
          ;ENDFOLD
          SLIN XP119 WITH $VEL = SVEL_CP(0.1, , LCPDAT28), $TOOL = STOOL2(FP119), $BASE = SBASE(FP119.BASE_NO), $IPO_MODE = SIPO_MODE(FP119.IPO_FRAME), $LOAD = SLOAD(FP119.TOOL_NO), $ACC = SACC_CP(LCPDAT28), $ORI_TYPE = SORI_TYP(LCPDAT28), $APO = SAPO(LCPDAT28), $JERK = SJERK(LCPDAT28), $COLLMON_TOL_PRO[1] = USE_CM_PRO_VALUES(0)
          ;ENDFOLD
          ;FOLD SPTP P600 Vel=100 % PDAT1 Tool[1]:SMC Base[0] ;%{PE}
          ;FOLD Parameters ;%{h}
          ;Params IlfProvider=kukaroboter.basistech.inlineforms.movement.spline; Kuka.IsGlobalPoint=False; Kuka.PointName=P600; Kuka.BlendingEnabled=False; Kuka.MoveDataPtpName=PDAT1; Kuka.VelocityPtp=100; Kuka.VelocityFieldEnabled=True; Kuka.ColDetectFieldEnabled=True; Kuka.CurrentCDSetIndex=0; Kuka.MovementParameterFieldEnabled=True; IlfCommand=SPTP
          ;ENDFOLD
          SPTP XP600 WITH $VEL_AXIS[1] = SVEL_JOINT(100.0), $TOOL = STOOL2(FP600), $BASE = SBASE(FP600.BASE_NO), $IPO_MODE = SIPO_MODE(FP600.IPO_FRAME), $LOAD = SLOAD(FP600.TOOL_NO), $ACC_AXIS[1] = SACC_JOINT(PPDAT1), $APO = SAPO_PTP(PPDAT1), $GEAR_JERK[1] = SGEAR_JERK(PPDAT1), $COLLMON_TOL_PRO[1] = USE_CM_PRO_VALUES(0)
          ;ENDFOLD
          ;FOLD SLIN P601 Vel=0.1 m/s CPDAT27 Tool[1]:SMC Base[0] ;%{PE}
          ;FOLD Parameters ;%{h}
          ;Params IlfProvider=kukaroboter.basistech.inlineforms.movement.spline; Kuka.IsGlobalPoint=False; Kuka.PointName=P601; Kuka.BlendingEnabled=False; Kuka.MoveDataName=CPDAT27; Kuka.VelocityPath=0.1; Kuka.VelocityFieldEnabled=True; Kuka.ColDetectFieldEnabled=True; Kuka.CurrentCDSetIndex=0; Kuka.MovementParameterFieldEnabled=True; IlfCommand=SLIN
          ;ENDFOLD
          SLIN XP601 WITH $VEL = SVEL_CP(0.1, , LCPDAT27), $TOOL = STOOL2(FP601), $BASE = SBASE(FP601.BASE_NO), $IPO_MODE = SIPO_MODE(FP601.IPO_FRAME), $LOAD = SLOAD(FP601.TOOL_NO), $ACC = SACC_CP(LCPDAT27), $ORI_TYPE = SORI_TYP(LCPDAT27), $APO = SAPO(LCPDAT27), $JERK = SJERK(LCPDAT27), $COLLMON_TOL_PRO[1] = USE_CM_PRO_VALUES(0)
          ;ENDFOLD
          ;FOLD SLIN P602 Vel=0.1 m/s CPDAT27 Tool[1]:SMC Base[0] ;%{PE}
          ;FOLD Parameters ;%{h}
          ;Params IlfProvider=kukaroboter.basistech.inlineforms.movement.spline; Kuka.IsGlobalPoint=False; Kuka.PointName=P602; Kuka.BlendingEnabled=False; Kuka.MoveDataName=CPDAT27; Kuka.VelocityPath=0.1; Kuka.VelocityFieldEnabled=True; Kuka.ColDetectFieldEnabled=True; Kuka.CurrentCDSetIndex=0; Kuka.MovementParameterFieldEnabled=True; IlfCommand=SLIN
          ;ENDFOLD
          SLIN XP602 WITH $VEL = SVEL_CP(0.1, , LCPDAT27), $TOOL = STOOL2(FP602), $BASE = SBASE(FP602.BASE_NO), $IPO_MODE = SIPO_MODE(FP602.IPO_FRAME), $LOAD = SLOAD(FP602.TOOL_NO), $ACC = SACC_CP(LCPDAT27), $ORI_TYPE = SORI_TYP(LCPDAT27), $APO = SAPO(LCPDAT27), $JERK = SJERK(LCPDAT27), $COLLMON_TOL_PRO[1] = USE_CM_PRO_VALUES(0)
          ;ENDFOLD
        ENDIF
        IF finalPosition == 20 THEN
          ;FOLD SPTP P120 Vel=100 % PDAT1 Tool[1]:SMC Base[0] ;%{PE}
          ;FOLD Parameters ;%{h}
          ;Params IlfProvider=kukaroboter.basistech.inlineforms.movement.spline; Kuka.IsGlobalPoint=False; Kuka.PointName=P120; Kuka.BlendingEnabled=False; Kuka.MoveDataPtpName=PDAT1; Kuka.VelocityPtp=100; Kuka.VelocityFieldEnabled=True; Kuka.ColDetectFieldEnabled=True; Kuka.CurrentCDSetIndex=0; Kuka.MovementParameterFieldEnabled=True; IlfCommand=SPTP
          ;ENDFOLD
          SPTP XP120 WITH $VEL_AXIS[1] = SVEL_JOINT(100.0), $TOOL = STOOL2(FP120), $BASE = SBASE(FP120.BASE_NO), $IPO_MODE = SIPO_MODE(FP120.IPO_FRAME), $LOAD = SLOAD(FP120.TOOL_NO), $ACC_AXIS[1] = SACC_JOINT(PPDAT1), $APO = SAPO_PTP(PPDAT1), $GEAR_JERK[1] = SGEAR_JERK(PPDAT1), $COLLMON_TOL_PRO[1] = USE_CM_PRO_VALUES(0)
          ;ENDFOLD
          ;FOLD SLIN P220 Vel=0.1 m/s CPDAT27 Tool[1]:SMC Base[0] ;%{PE}
          ;FOLD Parameters ;%{h}
          ;Params IlfProvider=kukaroboter.basistech.inlineforms.movement.spline; Kuka.IsGlobalPoint=False; Kuka.PointName=P220; Kuka.BlendingEnabled=False; Kuka.MoveDataName=CPDAT27; Kuka.VelocityPath=0.1; Kuka.VelocityFieldEnabled=True; Kuka.ColDetectFieldEnabled=True; Kuka.CurrentCDSetIndex=0; Kuka.MovementParameterFieldEnabled=True; IlfCommand=SLIN
          ;ENDFOLD
          SLIN XP220 WITH $VEL = SVEL_CP(0.1, , LCPDAT27), $TOOL = STOOL2(FP220), $BASE = SBASE(FP220.BASE_NO), $IPO_MODE = SIPO_MODE(FP220.IPO_FRAME), $LOAD = SLOAD(FP220.TOOL_NO), $ACC = SACC_CP(LCPDAT27), $ORI_TYPE = SORI_TYP(LCPDAT27), $APO = SAPO(LCPDAT27), $JERK = SJERK(LCPDAT27), $COLLMON_TOL_PRO[1] = USE_CM_PRO_VALUES(0)
          ;ENDFOLD
          ;FOLD Gripper SET [1]Gripper1 State=[1]ABIERTA Wait 0.2[s] Check with Strategy 1 ;%{PE}
          ;FOLD Parameters Parameters ;%{h}
          ;Params IlfProvider=GripperTech.GripperSet;setgripper=1;setstate=1;setcont=nocont;waittime=0.2;errorstrategy=1
          ;ENDFOLD
          GRPg_SetStateAndCheck(1, 1, 0.2, 1)
          ;ENDFOLD
          ;FOLD SLIN P120 Vel=0.1 m/s CPDAT28 Tool[1]:SMC Base[0] ;%{PE}
          ;FOLD Parameters ;%{h}
          ;Params IlfProvider=kukaroboter.basistech.inlineforms.movement.spline; Kuka.IsGlobalPoint=False; Kuka.PointName=P120; Kuka.BlendingEnabled=False; Kuka.MoveDataName=CPDAT28; Kuka.VelocityPath=0.1; Kuka.VelocityFieldEnabled=True; Kuka.ColDetectFieldEnabled=True; Kuka.CurrentCDSetIndex=0; Kuka.MovementParameterFieldEnabled=True; IlfCommand=SLIN
          ;ENDFOLD
          SLIN XP120 WITH $VEL = SVEL_CP(0.1, , LCPDAT28), $TOOL = STOOL2(FP120), $BASE = SBASE(FP120.BASE_NO), $IPO_MODE = SIPO_MODE(FP120.IPO_FRAME), $LOAD = SLOAD(FP120.TOOL_NO), $ACC = SACC_CP(LCPDAT28), $ORI_TYPE = SORI_TYP(LCPDAT28), $APO = SAPO(LCPDAT28), $JERK = SJERK(LCPDAT28), $COLLMON_TOL_PRO[1] = USE_CM_PRO_VALUES(0)
          ;ENDFOLD
          ;FOLD SPTP P600 Vel=100 % PDAT1 Tool[1]:SMC Base[0] ;%{PE}
          ;FOLD Parameters ;%{h}
          ;Params IlfProvider=kukaroboter.basistech.inlineforms.movement.spline; Kuka.IsGlobalPoint=False; Kuka.PointName=P600; Kuka.BlendingEnabled=False; Kuka.MoveDataPtpName=PDAT1; Kuka.VelocityPtp=100; Kuka.VelocityFieldEnabled=True; Kuka.ColDetectFieldEnabled=True; Kuka.CurrentCDSetIndex=0; Kuka.MovementParameterFieldEnabled=True; IlfCommand=SPTP
          ;ENDFOLD
          SPTP XP600 WITH $VEL_AXIS[1] = SVEL_JOINT(100.0), $TOOL = STOOL2(FP600), $BASE = SBASE(FP600.BASE_NO), $IPO_MODE = SIPO_MODE(FP600.IPO_FRAME), $LOAD = SLOAD(FP600.TOOL_NO), $ACC_AXIS[1] = SACC_JOINT(PPDAT1), $APO = SAPO_PTP(PPDAT1), $GEAR_JERK[1] = SGEAR_JERK(PPDAT1), $COLLMON_TOL_PRO[1] = USE_CM_PRO_VALUES(0)
          ;ENDFOLD
          ;FOLD SLIN P601 Vel=0.1 m/s CPDAT27 Tool[1]:SMC Base[0] ;%{PE}
          ;FOLD Parameters ;%{h}
          ;Params IlfProvider=kukaroboter.basistech.inlineforms.movement.spline; Kuka.IsGlobalPoint=False; Kuka.PointName=P601; Kuka.BlendingEnabled=False; Kuka.MoveDataName=CPDAT27; Kuka.VelocityPath=0.1; Kuka.VelocityFieldEnabled=True; Kuka.ColDetectFieldEnabled=True; Kuka.CurrentCDSetIndex=0; Kuka.MovementParameterFieldEnabled=True; IlfCommand=SLIN
          ;ENDFOLD
          SLIN XP601 WITH $VEL = SVEL_CP(0.1, , LCPDAT27), $TOOL = STOOL2(FP601), $BASE = SBASE(FP601.BASE_NO), $IPO_MODE = SIPO_MODE(FP601.IPO_FRAME), $LOAD = SLOAD(FP601.TOOL_NO), $ACC = SACC_CP(LCPDAT27), $ORI_TYPE = SORI_TYP(LCPDAT27), $APO = SAPO(LCPDAT27), $JERK = SJERK(LCPDAT27), $COLLMON_TOL_PRO[1] = USE_CM_PRO_VALUES(0)
          ;ENDFOLD
          ;FOLD SLIN P602 Vel=0.1 m/s CPDAT27 Tool[1]:SMC Base[0] ;%{PE}
          ;FOLD Parameters ;%{h}
          ;Params IlfProvider=kukaroboter.basistech.inlineforms.movement.spline; Kuka.IsGlobalPoint=False; Kuka.PointName=P602; Kuka.BlendingEnabled=False; Kuka.MoveDataName=CPDAT27; Kuka.VelocityPath=0.1; Kuka.VelocityFieldEnabled=True; Kuka.ColDetectFieldEnabled=True; Kuka.CurrentCDSetIndex=0; Kuka.MovementParameterFieldEnabled=True; IlfCommand=SLIN
          ;ENDFOLD
          SLIN XP602 WITH $VEL = SVEL_CP(0.1, , LCPDAT27), $TOOL = STOOL2(FP602), $BASE = SBASE(FP602.BASE_NO), $IPO_MODE = SIPO_MODE(FP602.IPO_FRAME), $LOAD = SLOAD(FP602.TOOL_NO), $ACC = SACC_CP(LCPDAT27), $ORI_TYPE = SORI_TYP(LCPDAT27), $APO = SAPO(LCPDAT27), $JERK = SJERK(LCPDAT27), $COLLMON_TOL_PRO[1] = USE_CM_PRO_VALUES(0)
          ;ENDFOLD
        ENDIF
        IF finalPosition == 21 THEN
          ;FOLD SPTP P121 Vel=100 % PDAT1 Tool[1]:SMC Base[0] ;%{PE}
          ;FOLD Parameters ;%{h}
          ;Params IlfProvider=kukaroboter.basistech.inlineforms.movement.spline; Kuka.IsGlobalPoint=False; Kuka.PointName=P121; Kuka.BlendingEnabled=False; Kuka.MoveDataPtpName=PDAT1; Kuka.VelocityPtp=100; Kuka.VelocityFieldEnabled=True; Kuka.ColDetectFieldEnabled=True; Kuka.CurrentCDSetIndex=0; Kuka.MovementParameterFieldEnabled=True; IlfCommand=SPTP
          ;ENDFOLD
          SPTP XP121 WITH $VEL_AXIS[1] = SVEL_JOINT(100.0), $TOOL = STOOL2(FP121), $BASE = SBASE(FP121.BASE_NO), $IPO_MODE = SIPO_MODE(FP121.IPO_FRAME), $LOAD = SLOAD(FP121.TOOL_NO), $ACC_AXIS[1] = SACC_JOINT(PPDAT1), $APO = SAPO_PTP(PPDAT1), $GEAR_JERK[1] = SGEAR_JERK(PPDAT1), $COLLMON_TOL_PRO[1] = USE_CM_PRO_VALUES(0)
          ;ENDFOLD
          ;FOLD SLIN P221 Vel=0.1 m/s CPDAT27 Tool[1]:SMC Base[0] ;%{PE}
          ;FOLD Parameters ;%{h}
          ;Params IlfProvider=kukaroboter.basistech.inlineforms.movement.spline; Kuka.IsGlobalPoint=False; Kuka.PointName=P221; Kuka.BlendingEnabled=False; Kuka.MoveDataName=CPDAT27; Kuka.VelocityPath=0.1; Kuka.VelocityFieldEnabled=True; Kuka.ColDetectFieldEnabled=True; Kuka.CurrentCDSetIndex=0; Kuka.MovementParameterFieldEnabled=True; IlfCommand=SLIN
          ;ENDFOLD
          SLIN XP221 WITH $VEL = SVEL_CP(0.1, , LCPDAT27), $TOOL = STOOL2(FP221), $BASE = SBASE(FP221.BASE_NO), $IPO_MODE = SIPO_MODE(FP221.IPO_FRAME), $LOAD = SLOAD(FP221.TOOL_NO), $ACC = SACC_CP(LCPDAT27), $ORI_TYPE = SORI_TYP(LCPDAT27), $APO = SAPO(LCPDAT27), $JERK = SJERK(LCPDAT27), $COLLMON_TOL_PRO[1] = USE_CM_PRO_VALUES(0)
          ;ENDFOLD
          ;FOLD Gripper SET [1]Gripper1 State=[1]ABIERTA Wait 0.2[s] Check with Strategy 1 ;%{PE}
          ;FOLD Parameters Parameters ;%{h}
          ;Params IlfProvider=GripperTech.GripperSet;setgripper=1;setstate=1;setcont=nocont;waittime=0.2;errorstrategy=1
          ;ENDFOLD
          GRPg_SetStateAndCheck(1, 1, 0.2, 1)
          ;ENDFOLD
          ;FOLD SLIN P121 Vel=0.1 m/s CPDAT28 Tool[1]:SMC Base[0] ;%{PE}
          ;FOLD Parameters ;%{h}
          ;Params IlfProvider=kukaroboter.basistech.inlineforms.movement.spline; Kuka.IsGlobalPoint=False; Kuka.PointName=P121; Kuka.BlendingEnabled=False; Kuka.MoveDataName=CPDAT28; Kuka.VelocityPath=0.1; Kuka.VelocityFieldEnabled=True; Kuka.ColDetectFieldEnabled=True; Kuka.CurrentCDSetIndex=0; Kuka.MovementParameterFieldEnabled=True; IlfCommand=SLIN
          ;ENDFOLD
          SLIN XP121 WITH $VEL = SVEL_CP(0.1, , LCPDAT28), $TOOL = STOOL2(FP121), $BASE = SBASE(FP121.BASE_NO), $IPO_MODE = SIPO_MODE(FP121.IPO_FRAME), $LOAD = SLOAD(FP121.TOOL_NO), $ACC = SACC_CP(LCPDAT28), $ORI_TYPE = SORI_TYP(LCPDAT28), $APO = SAPO(LCPDAT28), $JERK = SJERK(LCPDAT28), $COLLMON_TOL_PRO[1] = USE_CM_PRO_VALUES(0)
          ;ENDFOLD
          ;FOLD SPTP P600 Vel=100 % PDAT1 Tool[1]:SMC Base[0] ;%{PE}
          ;FOLD Parameters ;%{h}
          ;Params IlfProvider=kukaroboter.basistech.inlineforms.movement.spline; Kuka.IsGlobalPoint=False; Kuka.PointName=P600; Kuka.BlendingEnabled=False; Kuka.MoveDataPtpName=PDAT1; Kuka.VelocityPtp=100; Kuka.VelocityFieldEnabled=True; Kuka.ColDetectFieldEnabled=True; Kuka.CurrentCDSetIndex=0; Kuka.MovementParameterFieldEnabled=True; IlfCommand=SPTP
          ;ENDFOLD
          SPTP XP600 WITH $VEL_AXIS[1] = SVEL_JOINT(100.0), $TOOL = STOOL2(FP600), $BASE = SBASE(FP600.BASE_NO), $IPO_MODE = SIPO_MODE(FP600.IPO_FRAME), $LOAD = SLOAD(FP600.TOOL_NO), $ACC_AXIS[1] = SACC_JOINT(PPDAT1), $APO = SAPO_PTP(PPDAT1), $GEAR_JERK[1] = SGEAR_JERK(PPDAT1), $COLLMON_TOL_PRO[1] = USE_CM_PRO_VALUES(0)
          ;ENDFOLD
          ;FOLD SLIN P601 Vel=0.1 m/s CPDAT27 Tool[1]:SMC Base[0] ;%{PE}
          ;FOLD Parameters ;%{h}
          ;Params IlfProvider=kukaroboter.basistech.inlineforms.movement.spline; Kuka.IsGlobalPoint=False; Kuka.PointName=P601; Kuka.BlendingEnabled=False; Kuka.MoveDataName=CPDAT27; Kuka.VelocityPath=0.1; Kuka.VelocityFieldEnabled=True; Kuka.ColDetectFieldEnabled=True; Kuka.CurrentCDSetIndex=0; Kuka.MovementParameterFieldEnabled=True; IlfCommand=SLIN
          ;ENDFOLD
          SLIN XP601 WITH $VEL = SVEL_CP(0.1, , LCPDAT27), $TOOL = STOOL2(FP601), $BASE = SBASE(FP601.BASE_NO), $IPO_MODE = SIPO_MODE(FP601.IPO_FRAME), $LOAD = SLOAD(FP601.TOOL_NO), $ACC = SACC_CP(LCPDAT27), $ORI_TYPE = SORI_TYP(LCPDAT27), $APO = SAPO(LCPDAT27), $JERK = SJERK(LCPDAT27), $COLLMON_TOL_PRO[1] = USE_CM_PRO_VALUES(0)
          ;ENDFOLD
          ;FOLD SLIN P602 Vel=0.1 m/s CPDAT27 Tool[1]:SMC Base[0] ;%{PE}
          ;FOLD Parameters ;%{h}
          ;Params IlfProvider=kukaroboter.basistech.inlineforms.movement.spline; Kuka.IsGlobalPoint=False; Kuka.PointName=P602; Kuka.BlendingEnabled=False; Kuka.MoveDataName=CPDAT27; Kuka.VelocityPath=0.1; Kuka.VelocityFieldEnabled=True; Kuka.ColDetectFieldEnabled=True; Kuka.CurrentCDSetIndex=0; Kuka.MovementParameterFieldEnabled=True; IlfCommand=SLIN
          ;ENDFOLD
          SLIN XP602 WITH $VEL = SVEL_CP(0.1, , LCPDAT27), $TOOL = STOOL2(FP602), $BASE = SBASE(FP602.BASE_NO), $IPO_MODE = SIPO_MODE(FP602.IPO_FRAME), $LOAD = SLOAD(FP602.TOOL_NO), $ACC = SACC_CP(LCPDAT27), $ORI_TYPE = SORI_TYP(LCPDAT27), $APO = SAPO(LCPDAT27), $JERK = SJERK(LCPDAT27), $COLLMON_TOL_PRO[1] = USE_CM_PRO_VALUES(0)
          ;ENDFOLD
        ENDIF
        IF finalPosition == 22 THEN
          ;FOLD SPTP P122 Vel=100 % PDAT1 Tool[1]:SMC Base[0] ;%{PE}
          ;FOLD Parameters ;%{h}
          ;Params IlfProvider=kukaroboter.basistech.inlineforms.movement.spline; Kuka.IsGlobalPoint=False; Kuka.PointName=P122; Kuka.BlendingEnabled=False; Kuka.MoveDataPtpName=PDAT1; Kuka.VelocityPtp=100; Kuka.VelocityFieldEnabled=True; Kuka.ColDetectFieldEnabled=True; Kuka.CurrentCDSetIndex=0; Kuka.MovementParameterFieldEnabled=True; IlfCommand=SPTP
          ;ENDFOLD
          SPTP XP122 WITH $VEL_AXIS[1] = SVEL_JOINT(100.0), $TOOL = STOOL2(FP122), $BASE = SBASE(FP122.BASE_NO), $IPO_MODE = SIPO_MODE(FP122.IPO_FRAME), $LOAD = SLOAD(FP122.TOOL_NO), $ACC_AXIS[1] = SACC_JOINT(PPDAT1), $APO = SAPO_PTP(PPDAT1), $GEAR_JERK[1] = SGEAR_JERK(PPDAT1), $COLLMON_TOL_PRO[1] = USE_CM_PRO_VALUES(0)
          ;ENDFOLD
          ;FOLD SLIN P222 Vel=0.1 m/s CPDAT27 Tool[1]:SMC Base[0] ;%{PE}
          ;FOLD Parameters ;%{h}
          ;Params IlfProvider=kukaroboter.basistech.inlineforms.movement.spline; Kuka.IsGlobalPoint=False; Kuka.PointName=P222; Kuka.BlendingEnabled=False; Kuka.MoveDataName=CPDAT27; Kuka.VelocityPath=0.1; Kuka.VelocityFieldEnabled=True; Kuka.ColDetectFieldEnabled=True; Kuka.CurrentCDSetIndex=0; Kuka.MovementParameterFieldEnabled=True; IlfCommand=SLIN
          ;ENDFOLD
          SLIN XP222 WITH $VEL = SVEL_CP(0.1, , LCPDAT27), $TOOL = STOOL2(FP222), $BASE = SBASE(FP222.BASE_NO), $IPO_MODE = SIPO_MODE(FP222.IPO_FRAME), $LOAD = SLOAD(FP222.TOOL_NO), $ACC = SACC_CP(LCPDAT27), $ORI_TYPE = SORI_TYP(LCPDAT27), $APO = SAPO(LCPDAT27), $JERK = SJERK(LCPDAT27), $COLLMON_TOL_PRO[1] = USE_CM_PRO_VALUES(0)
          ;ENDFOLD
          ;FOLD Gripper SET [1]Gripper1 State=[1]ABIERTA Wait 0.2[s] Check with Strategy 1 ;%{PE}
          ;FOLD Parameters Parameters ;%{h}
          ;Params IlfProvider=GripperTech.GripperSet;setgripper=1;setstate=1;setcont=nocont;waittime=0.2;errorstrategy=1
          ;ENDFOLD
          GRPg_SetStateAndCheck(1, 1, 0.2, 1)
          ;ENDFOLD
          ;FOLD SLIN P122 Vel=0.1 m/s CPDAT28 Tool[1]:SMC Base[0] ;%{PE}
          ;FOLD Parameters ;%{h}
          ;Params IlfProvider=kukaroboter.basistech.inlineforms.movement.spline; Kuka.IsGlobalPoint=False; Kuka.PointName=P122; Kuka.BlendingEnabled=False; Kuka.MoveDataName=CPDAT28; Kuka.VelocityPath=0.1; Kuka.VelocityFieldEnabled=True; Kuka.ColDetectFieldEnabled=True; Kuka.CurrentCDSetIndex=0; Kuka.MovementParameterFieldEnabled=True; IlfCommand=SLIN
          ;ENDFOLD
          SLIN XP122 WITH $VEL = SVEL_CP(0.1, , LCPDAT28), $TOOL = STOOL2(FP122), $BASE = SBASE(FP122.BASE_NO), $IPO_MODE = SIPO_MODE(FP122.IPO_FRAME), $LOAD = SLOAD(FP122.TOOL_NO), $ACC = SACC_CP(LCPDAT28), $ORI_TYPE = SORI_TYP(LCPDAT28), $APO = SAPO(LCPDAT28), $JERK = SJERK(LCPDAT28), $COLLMON_TOL_PRO[1] = USE_CM_PRO_VALUES(0)
          ;ENDFOLD
          ;FOLD SPTP P600 Vel=100 % PDAT1 Tool[1]:SMC Base[0] ;%{PE}
          ;FOLD Parameters ;%{h}
          ;Params IlfProvider=kukaroboter.basistech.inlineforms.movement.spline; Kuka.IsGlobalPoint=False; Kuka.PointName=P600; Kuka.BlendingEnabled=False; Kuka.MoveDataPtpName=PDAT1; Kuka.VelocityPtp=100; Kuka.VelocityFieldEnabled=True; Kuka.ColDetectFieldEnabled=True; Kuka.CurrentCDSetIndex=0; Kuka.MovementParameterFieldEnabled=True; IlfCommand=SPTP
          ;ENDFOLD
          SPTP XP600 WITH $VEL_AXIS[1] = SVEL_JOINT(100.0), $TOOL = STOOL2(FP600), $BASE = SBASE(FP600.BASE_NO), $IPO_MODE = SIPO_MODE(FP600.IPO_FRAME), $LOAD = SLOAD(FP600.TOOL_NO), $ACC_AXIS[1] = SACC_JOINT(PPDAT1), $APO = SAPO_PTP(PPDAT1), $GEAR_JERK[1] = SGEAR_JERK(PPDAT1), $COLLMON_TOL_PRO[1] = USE_CM_PRO_VALUES(0)
          ;ENDFOLD
          ;FOLD SLIN P601 Vel=0.1 m/s CPDAT27 Tool[1]:SMC Base[0] ;%{PE}
          ;FOLD Parameters ;%{h}
          ;Params IlfProvider=kukaroboter.basistech.inlineforms.movement.spline; Kuka.IsGlobalPoint=False; Kuka.PointName=P601; Kuka.BlendingEnabled=False; Kuka.MoveDataName=CPDAT27; Kuka.VelocityPath=0.1; Kuka.VelocityFieldEnabled=True; Kuka.ColDetectFieldEnabled=True; Kuka.CurrentCDSetIndex=0; Kuka.MovementParameterFieldEnabled=True; IlfCommand=SLIN
          ;ENDFOLD
          SLIN XP601 WITH $VEL = SVEL_CP(0.1, , LCPDAT27), $TOOL = STOOL2(FP601), $BASE = SBASE(FP601.BASE_NO), $IPO_MODE = SIPO_MODE(FP601.IPO_FRAME), $LOAD = SLOAD(FP601.TOOL_NO), $ACC = SACC_CP(LCPDAT27), $ORI_TYPE = SORI_TYP(LCPDAT27), $APO = SAPO(LCPDAT27), $JERK = SJERK(LCPDAT27), $COLLMON_TOL_PRO[1] = USE_CM_PRO_VALUES(0)
          ;ENDFOLD
          ;FOLD SLIN P602 Vel=0.1 m/s CPDAT27 Tool[1]:SMC Base[0] ;%{PE}
          ;FOLD Parameters ;%{h}
          ;Params IlfProvider=kukaroboter.basistech.inlineforms.movement.spline; Kuka.IsGlobalPoint=False; Kuka.PointName=P602; Kuka.BlendingEnabled=False; Kuka.MoveDataName=CPDAT27; Kuka.VelocityPath=0.1; Kuka.VelocityFieldEnabled=True; Kuka.ColDetectFieldEnabled=True; Kuka.CurrentCDSetIndex=0; Kuka.MovementParameterFieldEnabled=True; IlfCommand=SLIN
          ;ENDFOLD
          SLIN XP602 WITH $VEL = SVEL_CP(0.1, , LCPDAT27), $TOOL = STOOL2(FP602), $BASE = SBASE(FP602.BASE_NO), $IPO_MODE = SIPO_MODE(FP602.IPO_FRAME), $LOAD = SLOAD(FP602.TOOL_NO), $ACC = SACC_CP(LCPDAT27), $ORI_TYPE = SORI_TYP(LCPDAT27), $APO = SAPO(LCPDAT27), $JERK = SJERK(LCPDAT27), $COLLMON_TOL_PRO[1] = USE_CM_PRO_VALUES(0)
          ;ENDFOLD
        ENDIF
        IF finalPosition == 23 THEN
          ;FOLD SPTP P123 Vel=100 % PDAT1 Tool[1]:SMC Base[0] ;%{PE}
          ;FOLD Parameters ;%{h}
          ;Params IlfProvider=kukaroboter.basistech.inlineforms.movement.spline; Kuka.IsGlobalPoint=False; Kuka.PointName=P123; Kuka.BlendingEnabled=False; Kuka.MoveDataPtpName=PDAT1; Kuka.VelocityPtp=100; Kuka.VelocityFieldEnabled=True; Kuka.ColDetectFieldEnabled=True; Kuka.CurrentCDSetIndex=0; Kuka.MovementParameterFieldEnabled=True; IlfCommand=SPTP
          ;ENDFOLD
          SPTP XP123 WITH $VEL_AXIS[1] = SVEL_JOINT(100.0), $TOOL = STOOL2(FP123), $BASE = SBASE(FP123.BASE_NO), $IPO_MODE = SIPO_MODE(FP123.IPO_FRAME), $LOAD = SLOAD(FP123.TOOL_NO), $ACC_AXIS[1] = SACC_JOINT(PPDAT1), $APO = SAPO_PTP(PPDAT1), $GEAR_JERK[1] = SGEAR_JERK(PPDAT1), $COLLMON_TOL_PRO[1] = USE_CM_PRO_VALUES(0)
          ;ENDFOLD
          ;FOLD SLIN P223 Vel=0.1 m/s CPDAT27 Tool[1]:SMC Base[0] ;%{PE}
          ;FOLD Parameters ;%{h}
          ;Params IlfProvider=kukaroboter.basistech.inlineforms.movement.spline; Kuka.IsGlobalPoint=False; Kuka.PointName=P223; Kuka.BlendingEnabled=False; Kuka.MoveDataName=CPDAT27; Kuka.VelocityPath=0.1; Kuka.VelocityFieldEnabled=True; Kuka.ColDetectFieldEnabled=True; Kuka.CurrentCDSetIndex=0; Kuka.MovementParameterFieldEnabled=True; IlfCommand=SLIN
          ;ENDFOLD
          SLIN XP223 WITH $VEL = SVEL_CP(0.1, , LCPDAT27), $TOOL = STOOL2(FP223), $BASE = SBASE(FP223.BASE_NO), $IPO_MODE = SIPO_MODE(FP223.IPO_FRAME), $LOAD = SLOAD(FP223.TOOL_NO), $ACC = SACC_CP(LCPDAT27), $ORI_TYPE = SORI_TYP(LCPDAT27), $APO = SAPO(LCPDAT27), $JERK = SJERK(LCPDAT27), $COLLMON_TOL_PRO[1] = USE_CM_PRO_VALUES(0)
          ;ENDFOLD
          ;FOLD Gripper SET [1]Gripper1 State=[1]ABIERTA Wait 0.2[s] Check with Strategy 1 ;%{PE}
          ;FOLD Parameters Parameters ;%{h}
          ;Params IlfProvider=GripperTech.GripperSet;setgripper=1;setstate=1;setcont=nocont;waittime=0.2;errorstrategy=1
          ;ENDFOLD
          GRPg_SetStateAndCheck(1, 1, 0.2, 1)
          ;ENDFOLD
          ;FOLD SLIN P123 Vel=0.1 m/s CPDAT28 Tool[1]:SMC Base[0] ;%{PE}
          ;FOLD Parameters ;%{h}
          ;Params IlfProvider=kukaroboter.basistech.inlineforms.movement.spline; Kuka.IsGlobalPoint=False; Kuka.PointName=P123; Kuka.BlendingEnabled=False; Kuka.MoveDataName=CPDAT28; Kuka.VelocityPath=0.1; Kuka.VelocityFieldEnabled=True; Kuka.ColDetectFieldEnabled=True; Kuka.CurrentCDSetIndex=0; Kuka.MovementParameterFieldEnabled=True; IlfCommand=SLIN
          ;ENDFOLD
          SLIN XP123 WITH $VEL = SVEL_CP(0.1, , LCPDAT28), $TOOL = STOOL2(FP123), $BASE = SBASE(FP123.BASE_NO), $IPO_MODE = SIPO_MODE(FP123.IPO_FRAME), $LOAD = SLOAD(FP123.TOOL_NO), $ACC = SACC_CP(LCPDAT28), $ORI_TYPE = SORI_TYP(LCPDAT28), $APO = SAPO(LCPDAT28), $JERK = SJERK(LCPDAT28), $COLLMON_TOL_PRO[1] = USE_CM_PRO_VALUES(0)
          ;ENDFOLD
          ;FOLD SPTP P600 Vel=100 % PDAT1 Tool[1]:SMC Base[0] ;%{PE}
          ;FOLD Parameters ;%{h}
          ;Params IlfProvider=kukaroboter.basistech.inlineforms.movement.spline; Kuka.IsGlobalPoint=False; Kuka.PointName=P600; Kuka.BlendingEnabled=False; Kuka.MoveDataPtpName=PDAT1; Kuka.VelocityPtp=100; Kuka.VelocityFieldEnabled=True; Kuka.ColDetectFieldEnabled=True; Kuka.CurrentCDSetIndex=0; Kuka.MovementParameterFieldEnabled=True; IlfCommand=SPTP
          ;ENDFOLD
          SPTP XP600 WITH $VEL_AXIS[1] = SVEL_JOINT(100.0), $TOOL = STOOL2(FP600), $BASE = SBASE(FP600.BASE_NO), $IPO_MODE = SIPO_MODE(FP600.IPO_FRAME), $LOAD = SLOAD(FP600.TOOL_NO), $ACC_AXIS[1] = SACC_JOINT(PPDAT1), $APO = SAPO_PTP(PPDAT1), $GEAR_JERK[1] = SGEAR_JERK(PPDAT1), $COLLMON_TOL_PRO[1] = USE_CM_PRO_VALUES(0)
          ;ENDFOLD
          ;FOLD SLIN P601 Vel=0.1 m/s CPDAT27 Tool[1]:SMC Base[0] ;%{PE}
          ;FOLD Parameters ;%{h}
          ;Params IlfProvider=kukaroboter.basistech.inlineforms.movement.spline; Kuka.IsGlobalPoint=False; Kuka.PointName=P601; Kuka.BlendingEnabled=False; Kuka.MoveDataName=CPDAT27; Kuka.VelocityPath=0.1; Kuka.VelocityFieldEnabled=True; Kuka.ColDetectFieldEnabled=True; Kuka.CurrentCDSetIndex=0; Kuka.MovementParameterFieldEnabled=True; IlfCommand=SLIN
          ;ENDFOLD
          SLIN XP601 WITH $VEL = SVEL_CP(0.1, , LCPDAT27), $TOOL = STOOL2(FP601), $BASE = SBASE(FP601.BASE_NO), $IPO_MODE = SIPO_MODE(FP601.IPO_FRAME), $LOAD = SLOAD(FP601.TOOL_NO), $ACC = SACC_CP(LCPDAT27), $ORI_TYPE = SORI_TYP(LCPDAT27), $APO = SAPO(LCPDAT27), $JERK = SJERK(LCPDAT27), $COLLMON_TOL_PRO[1] = USE_CM_PRO_VALUES(0)
          ;ENDFOLD
          ;FOLD SLIN P602 Vel=0.1 m/s CPDAT27 Tool[1]:SMC Base[0] ;%{PE}
          ;FOLD Parameters ;%{h}
          ;Params IlfProvider=kukaroboter.basistech.inlineforms.movement.spline; Kuka.IsGlobalPoint=False; Kuka.PointName=P602; Kuka.BlendingEnabled=False; Kuka.MoveDataName=CPDAT27; Kuka.VelocityPath=0.1; Kuka.VelocityFieldEnabled=True; Kuka.ColDetectFieldEnabled=True; Kuka.CurrentCDSetIndex=0; Kuka.MovementParameterFieldEnabled=True; IlfCommand=SLIN
          ;ENDFOLD
          SLIN XP602 WITH $VEL = SVEL_CP(0.1, , LCPDAT27), $TOOL = STOOL2(FP602), $BASE = SBASE(FP602.BASE_NO), $IPO_MODE = SIPO_MODE(FP602.IPO_FRAME), $LOAD = SLOAD(FP602.TOOL_NO), $ACC = SACC_CP(LCPDAT27), $ORI_TYPE = SORI_TYP(LCPDAT27), $APO = SAPO(LCPDAT27), $JERK = SJERK(LCPDAT27), $COLLMON_TOL_PRO[1] = USE_CM_PRO_VALUES(0)
          ;ENDFOLD
        ENDIF
        IF finalPosition == 24 THEN
          ;FOLD SPTP P124 Vel=100 % PDAT1 Tool[1]:SMC Base[0] ;%{PE}
          ;FOLD Parameters ;%{h}
          ;Params IlfProvider=kukaroboter.basistech.inlineforms.movement.spline; Kuka.IsGlobalPoint=False; Kuka.PointName=P124; Kuka.BlendingEnabled=False; Kuka.MoveDataPtpName=PDAT1; Kuka.VelocityPtp=100; Kuka.VelocityFieldEnabled=True; Kuka.ColDetectFieldEnabled=True; Kuka.CurrentCDSetIndex=0; Kuka.MovementParameterFieldEnabled=True; IlfCommand=SPTP
          ;ENDFOLD
          SPTP XP124 WITH $VEL_AXIS[1] = SVEL_JOINT(100.0), $TOOL = STOOL2(FP124), $BASE = SBASE(FP124.BASE_NO), $IPO_MODE = SIPO_MODE(FP124.IPO_FRAME), $LOAD = SLOAD(FP124.TOOL_NO), $ACC_AXIS[1] = SACC_JOINT(PPDAT1), $APO = SAPO_PTP(PPDAT1), $GEAR_JERK[1] = SGEAR_JERK(PPDAT1), $COLLMON_TOL_PRO[1] = USE_CM_PRO_VALUES(0)
          ;ENDFOLD
          ;FOLD SLIN P224 Vel=0.1 m/s CPDAT27 Tool[1]:SMC Base[0] ;%{PE}
          ;FOLD Parameters ;%{h}
          ;Params IlfProvider=kukaroboter.basistech.inlineforms.movement.spline; Kuka.IsGlobalPoint=False; Kuka.PointName=P224; Kuka.BlendingEnabled=False; Kuka.MoveDataName=CPDAT27; Kuka.VelocityPath=0.1; Kuka.VelocityFieldEnabled=True; Kuka.ColDetectFieldEnabled=True; Kuka.CurrentCDSetIndex=0; Kuka.MovementParameterFieldEnabled=True; IlfCommand=SLIN
          ;ENDFOLD
          SLIN XP224 WITH $VEL = SVEL_CP(0.1, , LCPDAT27), $TOOL = STOOL2(FP224), $BASE = SBASE(FP224.BASE_NO), $IPO_MODE = SIPO_MODE(FP224.IPO_FRAME), $LOAD = SLOAD(FP224.TOOL_NO), $ACC = SACC_CP(LCPDAT27), $ORI_TYPE = SORI_TYP(LCPDAT27), $APO = SAPO(LCPDAT27), $JERK = SJERK(LCPDAT27), $COLLMON_TOL_PRO[1] = USE_CM_PRO_VALUES(0)
          ;ENDFOLD
          ;FOLD Gripper SET [1]Gripper1 State=[1]ABIERTA Wait 0.2[s] Check with Strategy 1 ;%{PE}
          ;FOLD Parameters Parameters ;%{h}
          ;Params IlfProvider=GripperTech.GripperSet;setgripper=1;setstate=1;setcont=nocont;waittime=0.2;errorstrategy=1
          ;ENDFOLD
          GRPg_SetStateAndCheck(1, 1, 0.2, 1)
          ;ENDFOLD
          ;FOLD SLIN P124 Vel=0.1 m/s CPDAT28 Tool[1]:SMC Base[0] ;%{PE}
          ;FOLD Parameters ;%{h}
          ;Params IlfProvider=kukaroboter.basistech.inlineforms.movement.spline; Kuka.IsGlobalPoint=False; Kuka.PointName=P124; Kuka.BlendingEnabled=False; Kuka.MoveDataName=CPDAT28; Kuka.VelocityPath=0.1; Kuka.VelocityFieldEnabled=True; Kuka.ColDetectFieldEnabled=True; Kuka.CurrentCDSetIndex=0; Kuka.MovementParameterFieldEnabled=True; IlfCommand=SLIN
          ;ENDFOLD
          SLIN XP124 WITH $VEL = SVEL_CP(0.1, , LCPDAT28), $TOOL = STOOL2(FP124), $BASE = SBASE(FP124.BASE_NO), $IPO_MODE = SIPO_MODE(FP124.IPO_FRAME), $LOAD = SLOAD(FP124.TOOL_NO), $ACC = SACC_CP(LCPDAT28), $ORI_TYPE = SORI_TYP(LCPDAT28), $APO = SAPO(LCPDAT28), $JERK = SJERK(LCPDAT28), $COLLMON_TOL_PRO[1] = USE_CM_PRO_VALUES(0)
          ;ENDFOLD
          ;FOLD SPTP P600 Vel=100 % PDAT1 Tool[1]:SMC Base[0] ;%{PE}
          ;FOLD Parameters ;%{h}
          ;Params IlfProvider=kukaroboter.basistech.inlineforms.movement.spline; Kuka.IsGlobalPoint=False; Kuka.PointName=P600; Kuka.BlendingEnabled=False; Kuka.MoveDataPtpName=PDAT1; Kuka.VelocityPtp=100; Kuka.VelocityFieldEnabled=True; Kuka.ColDetectFieldEnabled=True; Kuka.CurrentCDSetIndex=0; Kuka.MovementParameterFieldEnabled=True; IlfCommand=SPTP
          ;ENDFOLD
          SPTP XP600 WITH $VEL_AXIS[1] = SVEL_JOINT(100.0), $TOOL = STOOL2(FP600), $BASE = SBASE(FP600.BASE_NO), $IPO_MODE = SIPO_MODE(FP600.IPO_FRAME), $LOAD = SLOAD(FP600.TOOL_NO), $ACC_AXIS[1] = SACC_JOINT(PPDAT1), $APO = SAPO_PTP(PPDAT1), $GEAR_JERK[1] = SGEAR_JERK(PPDAT1), $COLLMON_TOL_PRO[1] = USE_CM_PRO_VALUES(0)
          ;ENDFOLD
          ;FOLD SLIN P601 Vel=0.1 m/s CPDAT27 Tool[1]:SMC Base[0] ;%{PE}
          ;FOLD Parameters ;%{h}
          ;Params IlfProvider=kukaroboter.basistech.inlineforms.movement.spline; Kuka.IsGlobalPoint=False; Kuka.PointName=P601; Kuka.BlendingEnabled=False; Kuka.MoveDataName=CPDAT27; Kuka.VelocityPath=0.1; Kuka.VelocityFieldEnabled=True; Kuka.ColDetectFieldEnabled=True; Kuka.CurrentCDSetIndex=0; Kuka.MovementParameterFieldEnabled=True; IlfCommand=SLIN
          ;ENDFOLD
          SLIN XP601 WITH $VEL = SVEL_CP(0.1, , LCPDAT27), $TOOL = STOOL2(FP601), $BASE = SBASE(FP601.BASE_NO), $IPO_MODE = SIPO_MODE(FP601.IPO_FRAME), $LOAD = SLOAD(FP601.TOOL_NO), $ACC = SACC_CP(LCPDAT27), $ORI_TYPE = SORI_TYP(LCPDAT27), $APO = SAPO(LCPDAT27), $JERK = SJERK(LCPDAT27), $COLLMON_TOL_PRO[1] = USE_CM_PRO_VALUES(0)
          ;ENDFOLD
          ;FOLD SLIN P602 Vel=0.1 m/s CPDAT27 Tool[1]:SMC Base[0] ;%{PE}
          ;FOLD Parameters ;%{h}
          ;Params IlfProvider=kukaroboter.basistech.inlineforms.movement.spline; Kuka.IsGlobalPoint=False; Kuka.PointName=P602; Kuka.BlendingEnabled=False; Kuka.MoveDataName=CPDAT27; Kuka.VelocityPath=0.1; Kuka.VelocityFieldEnabled=True; Kuka.ColDetectFieldEnabled=True; Kuka.CurrentCDSetIndex=0; Kuka.MovementParameterFieldEnabled=True; IlfCommand=SLIN
          ;ENDFOLD
          SLIN XP602 WITH $VEL = SVEL_CP(0.1, , LCPDAT27), $TOOL = STOOL2(FP602), $BASE = SBASE(FP602.BASE_NO), $IPO_MODE = SIPO_MODE(FP602.IPO_FRAME), $LOAD = SLOAD(FP602.TOOL_NO), $ACC = SACC_CP(LCPDAT27), $ORI_TYPE = SORI_TYP(LCPDAT27), $APO = SAPO(LCPDAT27), $JERK = SJERK(LCPDAT27), $COLLMON_TOL_PRO[1] = USE_CM_PRO_VALUES(0)
          ;ENDFOLD
        ENDIF
        IF finalPosition == 25 THEN
          ;FOLD SPTP P125 Vel=100 % PDAT1 Tool[1]:SMC Base[0] ;%{PE}
          ;FOLD Parameters ;%{h}
          ;Params IlfProvider=kukaroboter.basistech.inlineforms.movement.spline; Kuka.IsGlobalPoint=False; Kuka.PointName=P125; Kuka.BlendingEnabled=False; Kuka.MoveDataPtpName=PDAT1; Kuka.VelocityPtp=100; Kuka.VelocityFieldEnabled=True; Kuka.ColDetectFieldEnabled=True; Kuka.CurrentCDSetIndex=0; Kuka.MovementParameterFieldEnabled=True; IlfCommand=SPTP
          ;ENDFOLD
          SPTP XP125 WITH $VEL_AXIS[1] = SVEL_JOINT(100.0), $TOOL = STOOL2(FP125), $BASE = SBASE(FP125.BASE_NO), $IPO_MODE = SIPO_MODE(FP125.IPO_FRAME), $LOAD = SLOAD(FP125.TOOL_NO), $ACC_AXIS[1] = SACC_JOINT(PPDAT1), $APO = SAPO_PTP(PPDAT1), $GEAR_JERK[1] = SGEAR_JERK(PPDAT1), $COLLMON_TOL_PRO[1] = USE_CM_PRO_VALUES(0)
          ;ENDFOLD
          ;FOLD SLIN P225 Vel=0.1 m/s CPDAT27 Tool[1]:SMC Base[0] ;%{PE}
          ;FOLD Parameters ;%{h}
          ;Params IlfProvider=kukaroboter.basistech.inlineforms.movement.spline; Kuka.IsGlobalPoint=False; Kuka.PointName=P225; Kuka.BlendingEnabled=False; Kuka.MoveDataName=CPDAT27; Kuka.VelocityPath=0.1; Kuka.VelocityFieldEnabled=True; Kuka.ColDetectFieldEnabled=True; Kuka.CurrentCDSetIndex=0; Kuka.MovementParameterFieldEnabled=True; IlfCommand=SLIN
          ;ENDFOLD
          SLIN XP225 WITH $VEL = SVEL_CP(0.1, , LCPDAT27), $TOOL = STOOL2(FP225), $BASE = SBASE(FP225.BASE_NO), $IPO_MODE = SIPO_MODE(FP225.IPO_FRAME), $LOAD = SLOAD(FP225.TOOL_NO), $ACC = SACC_CP(LCPDAT27), $ORI_TYPE = SORI_TYP(LCPDAT27), $APO = SAPO(LCPDAT27), $JERK = SJERK(LCPDAT27), $COLLMON_TOL_PRO[1] = USE_CM_PRO_VALUES(0)
          ;ENDFOLD
          ;FOLD Gripper SET [1]Gripper1 State=[1]ABIERTA Wait 0.2[s] Check with Strategy 1 ;%{PE}
          ;FOLD Parameters Parameters ;%{h}
          ;Params IlfProvider=GripperTech.GripperSet;setgripper=1;setstate=1;setcont=nocont;waittime=0.2;errorstrategy=1
          ;ENDFOLD
          GRPg_SetStateAndCheck(1, 1, 0.2, 1)
          ;ENDFOLD
          ;FOLD SLIN P125 Vel=0.1 m/s CPDAT28 Tool[1]:SMC Base[0] ;%{PE}
          ;FOLD Parameters ;%{h}
          ;Params IlfProvider=kukaroboter.basistech.inlineforms.movement.spline; Kuka.IsGlobalPoint=False; Kuka.PointName=P125; Kuka.BlendingEnabled=False; Kuka.MoveDataName=CPDAT28; Kuka.VelocityPath=0.1; Kuka.VelocityFieldEnabled=True; Kuka.ColDetectFieldEnabled=True; Kuka.CurrentCDSetIndex=0; Kuka.MovementParameterFieldEnabled=True; IlfCommand=SLIN
          ;ENDFOLD
          SLIN XP125 WITH $VEL = SVEL_CP(0.1, , LCPDAT28), $TOOL = STOOL2(FP125), $BASE = SBASE(FP125.BASE_NO), $IPO_MODE = SIPO_MODE(FP125.IPO_FRAME), $LOAD = SLOAD(FP125.TOOL_NO), $ACC = SACC_CP(LCPDAT28), $ORI_TYPE = SORI_TYP(LCPDAT28), $APO = SAPO(LCPDAT28), $JERK = SJERK(LCPDAT28), $COLLMON_TOL_PRO[1] = USE_CM_PRO_VALUES(0)
          ;ENDFOLD
          ;FOLD SPTP P600 Vel=100 % PDAT1 Tool[1]:SMC Base[0] ;%{PE}
          ;FOLD Parameters ;%{h}
          ;Params IlfProvider=kukaroboter.basistech.inlineforms.movement.spline; Kuka.IsGlobalPoint=False; Kuka.PointName=P600; Kuka.BlendingEnabled=False; Kuka.MoveDataPtpName=PDAT1; Kuka.VelocityPtp=100; Kuka.VelocityFieldEnabled=True; Kuka.ColDetectFieldEnabled=True; Kuka.CurrentCDSetIndex=0; Kuka.MovementParameterFieldEnabled=True; IlfCommand=SPTP
          ;ENDFOLD
          SPTP XP600 WITH $VEL_AXIS[1] = SVEL_JOINT(100.0), $TOOL = STOOL2(FP600), $BASE = SBASE(FP600.BASE_NO), $IPO_MODE = SIPO_MODE(FP600.IPO_FRAME), $LOAD = SLOAD(FP600.TOOL_NO), $ACC_AXIS[1] = SACC_JOINT(PPDAT1), $APO = SAPO_PTP(PPDAT1), $GEAR_JERK[1] = SGEAR_JERK(PPDAT1), $COLLMON_TOL_PRO[1] = USE_CM_PRO_VALUES(0)
          ;ENDFOLD
          ;FOLD SLIN P601 Vel=0.1 m/s CPDAT27 Tool[1]:SMC Base[0] ;%{PE}
          ;FOLD Parameters ;%{h}
          ;Params IlfProvider=kukaroboter.basistech.inlineforms.movement.spline; Kuka.IsGlobalPoint=False; Kuka.PointName=P601; Kuka.BlendingEnabled=False; Kuka.MoveDataName=CPDAT27; Kuka.VelocityPath=0.1; Kuka.VelocityFieldEnabled=True; Kuka.ColDetectFieldEnabled=True; Kuka.CurrentCDSetIndex=0; Kuka.MovementParameterFieldEnabled=True; IlfCommand=SLIN
          ;ENDFOLD
          SLIN XP601 WITH $VEL = SVEL_CP(0.1, , LCPDAT27), $TOOL = STOOL2(FP601), $BASE = SBASE(FP601.BASE_NO), $IPO_MODE = SIPO_MODE(FP601.IPO_FRAME), $LOAD = SLOAD(FP601.TOOL_NO), $ACC = SACC_CP(LCPDAT27), $ORI_TYPE = SORI_TYP(LCPDAT27), $APO = SAPO(LCPDAT27), $JERK = SJERK(LCPDAT27), $COLLMON_TOL_PRO[1] = USE_CM_PRO_VALUES(0)
          ;ENDFOLD
          ;FOLD SLIN P602 Vel=0.1 m/s CPDAT27 Tool[1]:SMC Base[0] ;%{PE}
          ;FOLD Parameters ;%{h}
          ;Params IlfProvider=kukaroboter.basistech.inlineforms.movement.spline; Kuka.IsGlobalPoint=False; Kuka.PointName=P602; Kuka.BlendingEnabled=False; Kuka.MoveDataName=CPDAT27; Kuka.VelocityPath=0.1; Kuka.VelocityFieldEnabled=True; Kuka.ColDetectFieldEnabled=True; Kuka.CurrentCDSetIndex=0; Kuka.MovementParameterFieldEnabled=True; IlfCommand=SLIN
          ;ENDFOLD
          SLIN XP602 WITH $VEL = SVEL_CP(0.1, , LCPDAT27), $TOOL = STOOL2(FP602), $BASE = SBASE(FP602.BASE_NO), $IPO_MODE = SIPO_MODE(FP602.IPO_FRAME), $LOAD = SLOAD(FP602.TOOL_NO), $ACC = SACC_CP(LCPDAT27), $ORI_TYPE = SORI_TYP(LCPDAT27), $APO = SAPO(LCPDAT27), $JERK = SJERK(LCPDAT27), $COLLMON_TOL_PRO[1] = USE_CM_PRO_VALUES(0)
          ;ENDFOLD
        ENDIF


        IF finalPosition == 26 THEN
          ;FOLD SPTP P126 Vel=100 % PDAT1 Tool[1]:SMC Base[0] ;%{PE}
          ;FOLD Parameters ;%{h}
          ;Params IlfProvider=kukaroboter.basistech.inlineforms.movement.spline; Kuka.IsGlobalPoint=False; Kuka.PointName=P126; Kuka.BlendingEnabled=False; Kuka.MoveDataPtpName=PDAT1; Kuka.VelocityPtp=100; Kuka.VelocityFieldEnabled=True; Kuka.ColDetectFieldEnabled=True; Kuka.CurrentCDSetIndex=0; Kuka.MovementParameterFieldEnabled=True; IlfCommand=SPTP
          ;ENDFOLD
          SPTP XP126 WITH $VEL_AXIS[1] = SVEL_JOINT(100.0), $TOOL = STOOL2(FP126), $BASE = SBASE(FP126.BASE_NO), $IPO_MODE = SIPO_MODE(FP126.IPO_FRAME), $LOAD = SLOAD(FP126.TOOL_NO), $ACC_AXIS[1] = SACC_JOINT(PPDAT1), $APO = SAPO_PTP(PPDAT1), $GEAR_JERK[1] = SGEAR_JERK(PPDAT1), $COLLMON_TOL_PRO[1] = USE_CM_PRO_VALUES(0)
          ;ENDFOLD
          ;FOLD SLIN P226 Vel=0.1 m/s CPDAT27 Tool[1]:SMC Base[0] ;%{PE}
          ;FOLD Parameters ;%{h}
          ;Params IlfProvider=kukaroboter.basistech.inlineforms.movement.spline; Kuka.IsGlobalPoint=False; Kuka.PointName=P226; Kuka.BlendingEnabled=False; Kuka.MoveDataName=CPDAT27; Kuka.VelocityPath=0.1; Kuka.VelocityFieldEnabled=True; Kuka.ColDetectFieldEnabled=True; Kuka.CurrentCDSetIndex=0; Kuka.MovementParameterFieldEnabled=True; IlfCommand=SLIN
          ;ENDFOLD
          SLIN XP226 WITH $VEL = SVEL_CP(0.1, , LCPDAT27), $TOOL = STOOL2(FP226), $BASE = SBASE(FP226.BASE_NO), $IPO_MODE = SIPO_MODE(FP226.IPO_FRAME), $LOAD = SLOAD(FP226.TOOL_NO), $ACC = SACC_CP(LCPDAT27), $ORI_TYPE = SORI_TYP(LCPDAT27), $APO = SAPO(LCPDAT27), $JERK = SJERK(LCPDAT27), $COLLMON_TOL_PRO[1] = USE_CM_PRO_VALUES(0)
          ;ENDFOLD
          ;FOLD Gripper SET [1]Gripper1 State=[1]ABIERTA Wait 0.2[s] Check with Strategy 1 ;%{PE}
          ;FOLD Parameters Parameters ;%{h}
          ;Params IlfProvider=GripperTech.GripperSet;setgripper=1;setstate=1;setcont=nocont;waittime=0.2;errorstrategy=1
          ;ENDFOLD
          GRPg_SetStateAndCheck(1, 1, 0.2, 1)
          ;ENDFOLD
          ;FOLD SLIN P126 Vel=0.1 m/s CPDAT28 Tool[1]:SMC Base[0] ;%{PE}
          ;FOLD Parameters ;%{h}
          ;Params IlfProvider=kukaroboter.basistech.inlineforms.movement.spline; Kuka.IsGlobalPoint=False; Kuka.PointName=P126; Kuka.BlendingEnabled=False; Kuka.MoveDataName=CPDAT28; Kuka.VelocityPath=0.1; Kuka.VelocityFieldEnabled=True; Kuka.ColDetectFieldEnabled=True; Kuka.CurrentCDSetIndex=0; Kuka.MovementParameterFieldEnabled=True; IlfCommand=SLIN
          ;ENDFOLD
          SLIN XP126 WITH $VEL = SVEL_CP(0.1, , LCPDAT28), $TOOL = STOOL2(FP126), $BASE = SBASE(FP126.BASE_NO), $IPO_MODE = SIPO_MODE(FP126.IPO_FRAME), $LOAD = SLOAD(FP126.TOOL_NO), $ACC = SACC_CP(LCPDAT28), $ORI_TYPE = SORI_TYP(LCPDAT28), $APO = SAPO(LCPDAT28), $JERK = SJERK(LCPDAT28), $COLLMON_TOL_PRO[1] = USE_CM_PRO_VALUES(0)
          ;ENDFOLD
        ENDIF

        IF finalPosition == 27 THEN
          ;FOLD SPTP P127 Vel=100 % PDAT1 Tool[1]:SMC Base[0] ;%{PE}
          ;FOLD Parameters ;%{h}
          ;Params IlfProvider=kukaroboter.basistech.inlineforms.movement.spline; Kuka.IsGlobalPoint=False; Kuka.PointName=P127; Kuka.BlendingEnabled=False; Kuka.MoveDataPtpName=PDAT1; Kuka.VelocityPtp=100; Kuka.VelocityFieldEnabled=True; Kuka.ColDetectFieldEnabled=True; Kuka.CurrentCDSetIndex=0; Kuka.MovementParameterFieldEnabled=True; IlfCommand=SPTP
          ;ENDFOLD
          SPTP XP127 WITH $VEL_AXIS[1] = SVEL_JOINT(100.0), $TOOL = STOOL2(FP127), $BASE = SBASE(FP127.BASE_NO), $IPO_MODE = SIPO_MODE(FP127.IPO_FRAME), $LOAD = SLOAD(FP127.TOOL_NO), $ACC_AXIS[1] = SACC_JOINT(PPDAT1), $APO = SAPO_PTP(PPDAT1), $GEAR_JERK[1] = SGEAR_JERK(PPDAT1), $COLLMON_TOL_PRO[1] = USE_CM_PRO_VALUES(0)
          ;ENDFOLD
          ;FOLD SLIN P227 Vel=0.1 m/s CPDAT27 Tool[1]:SMC Base[0] ;%{PE}
          ;FOLD Parameters ;%{h}
          ;Params IlfProvider=kukaroboter.basistech.inlineforms.movement.spline; Kuka.IsGlobalPoint=False; Kuka.PointName=P227; Kuka.BlendingEnabled=False; Kuka.MoveDataName=CPDAT27; Kuka.VelocityPath=0.1; Kuka.VelocityFieldEnabled=True; Kuka.ColDetectFieldEnabled=True; Kuka.CurrentCDSetIndex=0; Kuka.MovementParameterFieldEnabled=True; IlfCommand=SLIN
          ;ENDFOLD
          SLIN XP227 WITH $VEL = SVEL_CP(0.1, , LCPDAT27), $TOOL = STOOL2(FP227), $BASE = SBASE(FP227.BASE_NO), $IPO_MODE = SIPO_MODE(FP227.IPO_FRAME), $LOAD = SLOAD(FP227.TOOL_NO), $ACC = SACC_CP(LCPDAT27), $ORI_TYPE = SORI_TYP(LCPDAT27), $APO = SAPO(LCPDAT27), $JERK = SJERK(LCPDAT27), $COLLMON_TOL_PRO[1] = USE_CM_PRO_VALUES(0)
          ;ENDFOLD
          ;FOLD Gripper SET [1]Gripper1 State=[1]ABIERTA Wait 0.2[s] Check with Strategy 1 ;%{PE}
          ;FOLD Parameters Parameters ;%{h}
          ;Params IlfProvider=GripperTech.GripperSet;setgripper=1;setstate=1;setcont=nocont;waittime=0.2;errorstrategy=1
          ;ENDFOLD
          GRPg_SetStateAndCheck(1, 1, 0.2, 1)
          ;ENDFOLD
          ;FOLD SLIN P127 Vel=0.1 m/s CPDAT28 Tool[1]:SMC Base[0] ;%{PE}
          ;FOLD Parameters ;%{h}
          ;Params IlfProvider=kukaroboter.basistech.inlineforms.movement.spline; Kuka.IsGlobalPoint=False; Kuka.PointName=P127; Kuka.BlendingEnabled=False; Kuka.MoveDataName=CPDAT28; Kuka.VelocityPath=0.1; Kuka.VelocityFieldEnabled=True; Kuka.ColDetectFieldEnabled=True; Kuka.CurrentCDSetIndex=0; Kuka.MovementParameterFieldEnabled=True; IlfCommand=SLIN
          ;ENDFOLD
          SLIN XP127 WITH $VEL = SVEL_CP(0.1, , LCPDAT28), $TOOL = STOOL2(FP127), $BASE = SBASE(FP127.BASE_NO), $IPO_MODE = SIPO_MODE(FP127.IPO_FRAME), $LOAD = SLOAD(FP127.TOOL_NO), $ACC = SACC_CP(LCPDAT28), $ORI_TYPE = SORI_TYP(LCPDAT28), $APO = SAPO(LCPDAT28), $JERK = SJERK(LCPDAT28), $COLLMON_TOL_PRO[1] = USE_CM_PRO_VALUES(0)
          ;ENDFOLD
          ;FOLD SPTP P600 Vel=100 % PDAT1 Tool[1]:SMC Base[0] ;%{PE}
          ;FOLD Parameters ;%{h}
          ;Params IlfProvider=kukaroboter.basistech.inlineforms.movement.spline; Kuka.IsGlobalPoint=False; Kuka.PointName=P600; Kuka.BlendingEnabled=False; Kuka.MoveDataPtpName=PDAT1; Kuka.VelocityPtp=100; Kuka.VelocityFieldEnabled=True; Kuka.ColDetectFieldEnabled=True; Kuka.CurrentCDSetIndex=0; Kuka.MovementParameterFieldEnabled=True; IlfCommand=SPTP
          ;ENDFOLD
          SPTP XP600 WITH $VEL_AXIS[1] = SVEL_JOINT(100.0), $TOOL = STOOL2(FP600), $BASE = SBASE(FP600.BASE_NO), $IPO_MODE = SIPO_MODE(FP600.IPO_FRAME), $LOAD = SLOAD(FP600.TOOL_NO), $ACC_AXIS[1] = SACC_JOINT(PPDAT1), $APO = SAPO_PTP(PPDAT1), $GEAR_JERK[1] = SGEAR_JERK(PPDAT1), $COLLMON_TOL_PRO[1] = USE_CM_PRO_VALUES(0)
          ;ENDFOLD
          ;FOLD SLIN P601 Vel=0.1 m/s CPDAT27 Tool[1]:SMC Base[0] ;%{PE}
          ;FOLD Parameters ;%{h}
          ;Params IlfProvider=kukaroboter.basistech.inlineforms.movement.spline; Kuka.IsGlobalPoint=False; Kuka.PointName=P601; Kuka.BlendingEnabled=False; Kuka.MoveDataName=CPDAT27; Kuka.VelocityPath=0.1; Kuka.VelocityFieldEnabled=True; Kuka.ColDetectFieldEnabled=True; Kuka.CurrentCDSetIndex=0; Kuka.MovementParameterFieldEnabled=True; IlfCommand=SLIN
          ;ENDFOLD
          SLIN XP601 WITH $VEL = SVEL_CP(0.1, , LCPDAT27), $TOOL = STOOL2(FP601), $BASE = SBASE(FP601.BASE_NO), $IPO_MODE = SIPO_MODE(FP601.IPO_FRAME), $LOAD = SLOAD(FP601.TOOL_NO), $ACC = SACC_CP(LCPDAT27), $ORI_TYPE = SORI_TYP(LCPDAT27), $APO = SAPO(LCPDAT27), $JERK = SJERK(LCPDAT27), $COLLMON_TOL_PRO[1] = USE_CM_PRO_VALUES(0)
          ;ENDFOLD
          ;FOLD SLIN P602 Vel=0.1 m/s CPDAT27 Tool[1]:SMC Base[0] ;%{PE}
          ;FOLD Parameters ;%{h}
          ;Params IlfProvider=kukaroboter.basistech.inlineforms.movement.spline; Kuka.IsGlobalPoint=False; Kuka.PointName=P602; Kuka.BlendingEnabled=False; Kuka.MoveDataName=CPDAT27; Kuka.VelocityPath=0.1; Kuka.VelocityFieldEnabled=True; Kuka.ColDetectFieldEnabled=True; Kuka.CurrentCDSetIndex=0; Kuka.MovementParameterFieldEnabled=True; IlfCommand=SLIN
          ;ENDFOLD
          SLIN XP602 WITH $VEL = SVEL_CP(0.1, , LCPDAT27), $TOOL = STOOL2(FP602), $BASE = SBASE(FP602.BASE_NO), $IPO_MODE = SIPO_MODE(FP602.IPO_FRAME), $LOAD = SLOAD(FP602.TOOL_NO), $ACC = SACC_CP(LCPDAT27), $ORI_TYPE = SORI_TYP(LCPDAT27), $APO = SAPO(LCPDAT27), $JERK = SJERK(LCPDAT27), $COLLMON_TOL_PRO[1] = USE_CM_PRO_VALUES(0)
          ;ENDFOLD
        ENDIF

        IF finalPosition == 28 THEN
          ;FOLD SPTP P128 Vel=100 % PDAT1 Tool[1]:SMC Base[0] ;%{PE}
          ;FOLD Parameters ;%{h}
          ;Params IlfProvider=kukaroboter.basistech.inlineforms.movement.spline; Kuka.IsGlobalPoint=False; Kuka.PointName=P128; Kuka.BlendingEnabled=False; Kuka.MoveDataPtpName=PDAT1; Kuka.VelocityPtp=100; Kuka.VelocityFieldEnabled=True; Kuka.ColDetectFieldEnabled=True; Kuka.CurrentCDSetIndex=0; Kuka.MovementParameterFieldEnabled=True; IlfCommand=SPTP
          ;ENDFOLD
          SPTP XP128 WITH $VEL_AXIS[1] = SVEL_JOINT(100.0), $TOOL = STOOL2(FP128), $BASE = SBASE(FP128.BASE_NO), $IPO_MODE = SIPO_MODE(FP128.IPO_FRAME), $LOAD = SLOAD(FP128.TOOL_NO), $ACC_AXIS[1] = SACC_JOINT(PPDAT1), $APO = SAPO_PTP(PPDAT1), $GEAR_JERK[1] = SGEAR_JERK(PPDAT1), $COLLMON_TOL_PRO[1] = USE_CM_PRO_VALUES(0)
          ;ENDFOLD
          ;FOLD SLIN P228 Vel=0.1 m/s CPDAT27 Tool[1]:SMC Base[0] ;%{PE}
          ;FOLD Parameters ;%{h}
          ;Params IlfProvider=kukaroboter.basistech.inlineforms.movement.spline; Kuka.IsGlobalPoint=False; Kuka.PointName=P228; Kuka.BlendingEnabled=False; Kuka.MoveDataName=CPDAT27; Kuka.VelocityPath=0.1; Kuka.VelocityFieldEnabled=True; Kuka.ColDetectFieldEnabled=True; Kuka.CurrentCDSetIndex=0; Kuka.MovementParameterFieldEnabled=True; IlfCommand=SLIN
          ;ENDFOLD
          SLIN XP228 WITH $VEL = SVEL_CP(0.1, , LCPDAT27), $TOOL = STOOL2(FP228), $BASE = SBASE(FP228.BASE_NO), $IPO_MODE = SIPO_MODE(FP228.IPO_FRAME), $LOAD = SLOAD(FP228.TOOL_NO), $ACC = SACC_CP(LCPDAT27), $ORI_TYPE = SORI_TYP(LCPDAT27), $APO = SAPO(LCPDAT27), $JERK = SJERK(LCPDAT27), $COLLMON_TOL_PRO[1] = USE_CM_PRO_VALUES(0)
          ;ENDFOLD
          ;FOLD Gripper SET [1]Gripper1 State=[1]ABIERTA Wait 0.2[s] Check with Strategy 1 ;%{PE}
          ;FOLD Parameters Parameters ;%{h}
          ;Params IlfProvider=GripperTech.GripperSet;setgripper=1;setstate=1;setcont=nocont;waittime=0.2;errorstrategy=1
          ;ENDFOLD
          GRPg_SetStateAndCheck(1, 1, 0.2, 1)
          ;ENDFOLD
          ;FOLD SLIN P128 Vel=0.1 m/s CPDAT28 Tool[1]:SMC Base[0] ;%{PE}
          ;FOLD Parameters ;%{h}
          ;Params IlfProvider=kukaroboter.basistech.inlineforms.movement.spline; Kuka.IsGlobalPoint=False; Kuka.PointName=P128; Kuka.BlendingEnabled=False; Kuka.MoveDataName=CPDAT28; Kuka.VelocityPath=0.1; Kuka.VelocityFieldEnabled=True; Kuka.ColDetectFieldEnabled=True; Kuka.CurrentCDSetIndex=0; Kuka.MovementParameterFieldEnabled=True; IlfCommand=SLIN
          ;ENDFOLD
          SLIN XP128 WITH $VEL = SVEL_CP(0.1, , LCPDAT28), $TOOL = STOOL2(FP128), $BASE = SBASE(FP128.BASE_NO), $IPO_MODE = SIPO_MODE(FP128.IPO_FRAME), $LOAD = SLOAD(FP128.TOOL_NO), $ACC = SACC_CP(LCPDAT28), $ORI_TYPE = SORI_TYP(LCPDAT28), $APO = SAPO(LCPDAT28), $JERK = SJERK(LCPDAT28), $COLLMON_TOL_PRO[1] = USE_CM_PRO_VALUES(0)
          ;ENDFOLD
          ;FOLD SPTP P600 Vel=100 % PDAT1 Tool[1]:SMC Base[0] ;%{PE}
          ;FOLD Parameters ;%{h}
          ;Params IlfProvider=kukaroboter.basistech.inlineforms.movement.spline; Kuka.IsGlobalPoint=False; Kuka.PointName=P600; Kuka.BlendingEnabled=False; Kuka.MoveDataPtpName=PDAT1; Kuka.VelocityPtp=100; Kuka.VelocityFieldEnabled=True; Kuka.ColDetectFieldEnabled=True; Kuka.CurrentCDSetIndex=0; Kuka.MovementParameterFieldEnabled=True; IlfCommand=SPTP
          ;ENDFOLD
          SPTP XP600 WITH $VEL_AXIS[1] = SVEL_JOINT(100.0), $TOOL = STOOL2(FP600), $BASE = SBASE(FP600.BASE_NO), $IPO_MODE = SIPO_MODE(FP600.IPO_FRAME), $LOAD = SLOAD(FP600.TOOL_NO), $ACC_AXIS[1] = SACC_JOINT(PPDAT1), $APO = SAPO_PTP(PPDAT1), $GEAR_JERK[1] = SGEAR_JERK(PPDAT1), $COLLMON_TOL_PRO[1] = USE_CM_PRO_VALUES(0)
          ;ENDFOLD
          ;FOLD SLIN P601 Vel=0.1 m/s CPDAT27 Tool[1]:SMC Base[0] ;%{PE}
          ;FOLD Parameters ;%{h}
          ;Params IlfProvider=kukaroboter.basistech.inlineforms.movement.spline; Kuka.IsGlobalPoint=False; Kuka.PointName=P601; Kuka.BlendingEnabled=False; Kuka.MoveDataName=CPDAT27; Kuka.VelocityPath=0.1; Kuka.VelocityFieldEnabled=True; Kuka.ColDetectFieldEnabled=True; Kuka.CurrentCDSetIndex=0; Kuka.MovementParameterFieldEnabled=True; IlfCommand=SLIN
          ;ENDFOLD
          SLIN XP601 WITH $VEL = SVEL_CP(0.1, , LCPDAT27), $TOOL = STOOL2(FP601), $BASE = SBASE(FP601.BASE_NO), $IPO_MODE = SIPO_MODE(FP601.IPO_FRAME), $LOAD = SLOAD(FP601.TOOL_NO), $ACC = SACC_CP(LCPDAT27), $ORI_TYPE = SORI_TYP(LCPDAT27), $APO = SAPO(LCPDAT27), $JERK = SJERK(LCPDAT27), $COLLMON_TOL_PRO[1] = USE_CM_PRO_VALUES(0)
          ;ENDFOLD
          ;FOLD SLIN P602 Vel=0.1 m/s CPDAT27 Tool[1]:SMC Base[0] ;%{PE}
          ;FOLD Parameters ;%{h}
          ;Params IlfProvider=kukaroboter.basistech.inlineforms.movement.spline; Kuka.IsGlobalPoint=False; Kuka.PointName=P602; Kuka.BlendingEnabled=False; Kuka.MoveDataName=CPDAT27; Kuka.VelocityPath=0.1; Kuka.VelocityFieldEnabled=True; Kuka.ColDetectFieldEnabled=True; Kuka.CurrentCDSetIndex=0; Kuka.MovementParameterFieldEnabled=True; IlfCommand=SLIN
          ;ENDFOLD
          SLIN XP602 WITH $VEL = SVEL_CP(0.1, , LCPDAT27), $TOOL = STOOL2(FP602), $BASE = SBASE(FP602.BASE_NO), $IPO_MODE = SIPO_MODE(FP602.IPO_FRAME), $LOAD = SLOAD(FP602.TOOL_NO), $ACC = SACC_CP(LCPDAT27), $ORI_TYPE = SORI_TYP(LCPDAT27), $APO = SAPO(LCPDAT27), $JERK = SJERK(LCPDAT27), $COLLMON_TOL_PRO[1] = USE_CM_PRO_VALUES(0)
          ;ENDFOLD
        ENDIF

        IF finalPosition == 29 THEN
          ;FOLD SPTP P129 Vel=100 % PDAT1 Tool[1]:SMC Base[0] ;%{PE}
          ;FOLD Parameters ;%{h}
          ;Params IlfProvider=kukaroboter.basistech.inlineforms.movement.spline; Kuka.IsGlobalPoint=False; Kuka.PointName=P129; Kuka.BlendingEnabled=False; Kuka.MoveDataPtpName=PDAT1; Kuka.VelocityPtp=100; Kuka.VelocityFieldEnabled=True; Kuka.ColDetectFieldEnabled=True; Kuka.CurrentCDSetIndex=0; Kuka.MovementParameterFieldEnabled=True; IlfCommand=SPTP
          ;ENDFOLD
          SPTP XP129 WITH $VEL_AXIS[1] = SVEL_JOINT(100.0), $TOOL = STOOL2(FP129), $BASE = SBASE(FP129.BASE_NO), $IPO_MODE = SIPO_MODE(FP129.IPO_FRAME), $LOAD = SLOAD(FP129.TOOL_NO), $ACC_AXIS[1] = SACC_JOINT(PPDAT1), $APO = SAPO_PTP(PPDAT1), $GEAR_JERK[1] = SGEAR_JERK(PPDAT1), $COLLMON_TOL_PRO[1] = USE_CM_PRO_VALUES(0)
          ;ENDFOLD
          ;FOLD SLIN P229 Vel=0.1 m/s CPDAT27 Tool[1]:SMC Base[0] ;%{PE}
          ;FOLD Parameters ;%{h}
          ;Params IlfProvider=kukaroboter.basistech.inlineforms.movement.spline; Kuka.IsGlobalPoint=False; Kuka.PointName=P229; Kuka.BlendingEnabled=False; Kuka.MoveDataName=CPDAT27; Kuka.VelocityPath=0.1; Kuka.VelocityFieldEnabled=True; Kuka.ColDetectFieldEnabled=True; Kuka.CurrentCDSetIndex=0; Kuka.MovementParameterFieldEnabled=True; IlfCommand=SLIN
          ;ENDFOLD
          SLIN XP229 WITH $VEL = SVEL_CP(0.1, , LCPDAT27), $TOOL = STOOL2(FP229), $BASE = SBASE(FP229.BASE_NO), $IPO_MODE = SIPO_MODE(FP229.IPO_FRAME), $LOAD = SLOAD(FP229.TOOL_NO), $ACC = SACC_CP(LCPDAT27), $ORI_TYPE = SORI_TYP(LCPDAT27), $APO = SAPO(LCPDAT27), $JERK = SJERK(LCPDAT27), $COLLMON_TOL_PRO[1] = USE_CM_PRO_VALUES(0)
          ;ENDFOLD
          ;FOLD Gripper SET [1]Gripper1 State=[1]ABIERTA Wait 0.2[s] Check with Strategy 1 ;%{PE}
          ;FOLD Parameters Parameters ;%{h}
          ;Params IlfProvider=GripperTech.GripperSet;setgripper=1;setstate=1;setcont=nocont;waittime=0.2;errorstrategy=1
          ;ENDFOLD
          GRPg_SetStateAndCheck(1, 1, 0.2, 1)
          ;ENDFOLD
          ;FOLD SLIN P129 Vel=0.1 m/s CPDAT28 Tool[1]:SMC Base[0] ;%{PE}
          ;FOLD Parameters ;%{h}
          ;Params IlfProvider=kukaroboter.basistech.inlineforms.movement.spline; Kuka.IsGlobalPoint=False; Kuka.PointName=P129; Kuka.BlendingEnabled=False; Kuka.MoveDataName=CPDAT28; Kuka.VelocityPath=0.1; Kuka.VelocityFieldEnabled=True; Kuka.ColDetectFieldEnabled=True; Kuka.CurrentCDSetIndex=0; Kuka.MovementParameterFieldEnabled=True; IlfCommand=SLIN
          ;ENDFOLD
          SLIN XP129 WITH $VEL = SVEL_CP(0.1, , LCPDAT28), $TOOL = STOOL2(FP129), $BASE = SBASE(FP129.BASE_NO), $IPO_MODE = SIPO_MODE(FP129.IPO_FRAME), $LOAD = SLOAD(FP129.TOOL_NO), $ACC = SACC_CP(LCPDAT28), $ORI_TYPE = SORI_TYP(LCPDAT28), $APO = SAPO(LCPDAT28), $JERK = SJERK(LCPDAT28), $COLLMON_TOL_PRO[1] = USE_CM_PRO_VALUES(0)
          ;ENDFOLD
          ;FOLD SPTP P600 Vel=100 % PDAT1 Tool[1]:SMC Base[0] ;%{PE}
          ;FOLD Parameters ;%{h}
          ;Params IlfProvider=kukaroboter.basistech.inlineforms.movement.spline; Kuka.IsGlobalPoint=False; Kuka.PointName=P600; Kuka.BlendingEnabled=False; Kuka.MoveDataPtpName=PDAT1; Kuka.VelocityPtp=100; Kuka.VelocityFieldEnabled=True; Kuka.ColDetectFieldEnabled=True; Kuka.CurrentCDSetIndex=0; Kuka.MovementParameterFieldEnabled=True; IlfCommand=SPTP
          ;ENDFOLD
          SPTP XP600 WITH $VEL_AXIS[1] = SVEL_JOINT(100.0), $TOOL = STOOL2(FP600), $BASE = SBASE(FP600.BASE_NO), $IPO_MODE = SIPO_MODE(FP600.IPO_FRAME), $LOAD = SLOAD(FP600.TOOL_NO), $ACC_AXIS[1] = SACC_JOINT(PPDAT1), $APO = SAPO_PTP(PPDAT1), $GEAR_JERK[1] = SGEAR_JERK(PPDAT1), $COLLMON_TOL_PRO[1] = USE_CM_PRO_VALUES(0)
          ;ENDFOLD
          ;FOLD SLIN P601 Vel=0.1 m/s CPDAT27 Tool[1]:SMC Base[0] ;%{PE}
          ;FOLD Parameters ;%{h}
          ;Params IlfProvider=kukaroboter.basistech.inlineforms.movement.spline; Kuka.IsGlobalPoint=False; Kuka.PointName=P601; Kuka.BlendingEnabled=False; Kuka.MoveDataName=CPDAT27; Kuka.VelocityPath=0.1; Kuka.VelocityFieldEnabled=True; Kuka.ColDetectFieldEnabled=True; Kuka.CurrentCDSetIndex=0; Kuka.MovementParameterFieldEnabled=True; IlfCommand=SLIN
          ;ENDFOLD
          SLIN XP601 WITH $VEL = SVEL_CP(0.1, , LCPDAT27), $TOOL = STOOL2(FP601), $BASE = SBASE(FP601.BASE_NO), $IPO_MODE = SIPO_MODE(FP601.IPO_FRAME), $LOAD = SLOAD(FP601.TOOL_NO), $ACC = SACC_CP(LCPDAT27), $ORI_TYPE = SORI_TYP(LCPDAT27), $APO = SAPO(LCPDAT27), $JERK = SJERK(LCPDAT27), $COLLMON_TOL_PRO[1] = USE_CM_PRO_VALUES(0)
          ;ENDFOLD
          ;FOLD SLIN P602 Vel=0.1 m/s CPDAT27 Tool[1]:SMC Base[0] ;%{PE}
          ;FOLD Parameters ;%{h}
          ;Params IlfProvider=kukaroboter.basistech.inlineforms.movement.spline; Kuka.IsGlobalPoint=False; Kuka.PointName=P602; Kuka.BlendingEnabled=False; Kuka.MoveDataName=CPDAT27; Kuka.VelocityPath=0.1; Kuka.VelocityFieldEnabled=True; Kuka.ColDetectFieldEnabled=True; Kuka.CurrentCDSetIndex=0; Kuka.MovementParameterFieldEnabled=True; IlfCommand=SLIN
          ;ENDFOLD
          SLIN XP602 WITH $VEL = SVEL_CP(0.1, , LCPDAT27), $TOOL = STOOL2(FP602), $BASE = SBASE(FP602.BASE_NO), $IPO_MODE = SIPO_MODE(FP602.IPO_FRAME), $LOAD = SLOAD(FP602.TOOL_NO), $ACC = SACC_CP(LCPDAT27), $ORI_TYPE = SORI_TYP(LCPDAT27), $APO = SAPO(LCPDAT27), $JERK = SJERK(LCPDAT27), $COLLMON_TOL_PRO[1] = USE_CM_PRO_VALUES(0)
          ;ENDFOLD
        ENDIF

        IF finalPosition == 30 THEN
          ;FOLD SPTP P130 Vel=100 % PDAT1 Tool[1]:SMC Base[0] ;%{PE}
          ;FOLD Parameters ;%{h}
          ;Params IlfProvider=kukaroboter.basistech.inlineforms.movement.spline; Kuka.IsGlobalPoint=False; Kuka.PointName=P130; Kuka.BlendingEnabled=False; Kuka.MoveDataPtpName=PDAT1; Kuka.VelocityPtp=100; Kuka.VelocityFieldEnabled=True; Kuka.ColDetectFieldEnabled=True; Kuka.CurrentCDSetIndex=0; Kuka.MovementParameterFieldEnabled=True; IlfCommand=SPTP
          ;ENDFOLD
          SPTP XP130 WITH $VEL_AXIS[1] = SVEL_JOINT(100.0), $TOOL = STOOL2(FP130), $BASE = SBASE(FP130.BASE_NO), $IPO_MODE = SIPO_MODE(FP130.IPO_FRAME), $LOAD = SLOAD(FP130.TOOL_NO), $ACC_AXIS[1] = SACC_JOINT(PPDAT1), $APO = SAPO_PTP(PPDAT1), $GEAR_JERK[1] = SGEAR_JERK(PPDAT1), $COLLMON_TOL_PRO[1] = USE_CM_PRO_VALUES(0)
          ;ENDFOLD
          ;FOLD SLIN P230 Vel=0.1 m/s CPDAT27 Tool[1]:SMC Base[0] ;%{PE}
          ;FOLD Parameters ;%{h}
          ;Params IlfProvider=kukaroboter.basistech.inlineforms.movement.spline; Kuka.IsGlobalPoint=False; Kuka.PointName=P230; Kuka.BlendingEnabled=False; Kuka.MoveDataName=CPDAT27; Kuka.VelocityPath=0.1; Kuka.VelocityFieldEnabled=True; Kuka.ColDetectFieldEnabled=True; Kuka.CurrentCDSetIndex=0; Kuka.MovementParameterFieldEnabled=True; IlfCommand=SLIN
          ;ENDFOLD
          SLIN XP230 WITH $VEL = SVEL_CP(0.1, , LCPDAT27), $TOOL = STOOL2(FP230), $BASE = SBASE(FP230.BASE_NO), $IPO_MODE = SIPO_MODE(FP230.IPO_FRAME), $LOAD = SLOAD(FP230.TOOL_NO), $ACC = SACC_CP(LCPDAT27), $ORI_TYPE = SORI_TYP(LCPDAT27), $APO = SAPO(LCPDAT27), $JERK = SJERK(LCPDAT27), $COLLMON_TOL_PRO[1] = USE_CM_PRO_VALUES(0)
          ;ENDFOLD
          ;FOLD Gripper SET [1]Gripper1 State=[1]ABIERTA Wait 0.2[s] Check with Strategy 1 ;%{PE}
          ;FOLD Parameters Parameters ;%{h}
          ;Params IlfProvider=GripperTech.GripperSet;setgripper=1;setstate=1;setcont=nocont;waittime=0.2;errorstrategy=1
          ;ENDFOLD
          GRPg_SetStateAndCheck(1, 1, 0.2, 1)
          ;ENDFOLD
          ;FOLD SLIN P130 Vel=0.1 m/s CPDAT28 Tool[1]:SMC Base[0] ;%{PE}
          ;FOLD Parameters ;%{h}
          ;Params IlfProvider=kukaroboter.basistech.inlineforms.movement.spline; Kuka.IsGlobalPoint=False; Kuka.PointName=P130; Kuka.BlendingEnabled=False; Kuka.MoveDataName=CPDAT28; Kuka.VelocityPath=0.1; Kuka.VelocityFieldEnabled=True; Kuka.ColDetectFieldEnabled=True; Kuka.CurrentCDSetIndex=0; Kuka.MovementParameterFieldEnabled=True; IlfCommand=SLIN
          ;ENDFOLD
          SLIN XP130 WITH $VEL = SVEL_CP(0.1, , LCPDAT28), $TOOL = STOOL2(FP130), $BASE = SBASE(FP130.BASE_NO), $IPO_MODE = SIPO_MODE(FP130.IPO_FRAME), $LOAD = SLOAD(FP130.TOOL_NO), $ACC = SACC_CP(LCPDAT28), $ORI_TYPE = SORI_TYP(LCPDAT28), $APO = SAPO(LCPDAT28), $JERK = SJERK(LCPDAT28), $COLLMON_TOL_PRO[1] = USE_CM_PRO_VALUES(0)
          ;ENDFOLD
          ;FOLD SPTP P600 Vel=100 % PDAT1 Tool[1]:SMC Base[0] ;%{PE}
          ;FOLD Parameters ;%{h}
          ;Params IlfProvider=kukaroboter.basistech.inlineforms.movement.spline; Kuka.IsGlobalPoint=False; Kuka.PointName=P600; Kuka.BlendingEnabled=False; Kuka.MoveDataPtpName=PDAT1; Kuka.VelocityPtp=100; Kuka.VelocityFieldEnabled=True; Kuka.ColDetectFieldEnabled=True; Kuka.CurrentCDSetIndex=0; Kuka.MovementParameterFieldEnabled=True; IlfCommand=SPTP
          ;ENDFOLD
          SPTP XP600 WITH $VEL_AXIS[1] = SVEL_JOINT(100.0), $TOOL = STOOL2(FP600), $BASE = SBASE(FP600.BASE_NO), $IPO_MODE = SIPO_MODE(FP600.IPO_FRAME), $LOAD = SLOAD(FP600.TOOL_NO), $ACC_AXIS[1] = SACC_JOINT(PPDAT1), $APO = SAPO_PTP(PPDAT1), $GEAR_JERK[1] = SGEAR_JERK(PPDAT1), $COLLMON_TOL_PRO[1] = USE_CM_PRO_VALUES(0)
          ;ENDFOLD
          ;FOLD SLIN P601 Vel=0.1 m/s CPDAT27 Tool[1]:SMC Base[0] ;%{PE}
          ;FOLD Parameters ;%{h}
          ;Params IlfProvider=kukaroboter.basistech.inlineforms.movement.spline; Kuka.IsGlobalPoint=False; Kuka.PointName=P601; Kuka.BlendingEnabled=False; Kuka.MoveDataName=CPDAT27; Kuka.VelocityPath=0.1; Kuka.VelocityFieldEnabled=True; Kuka.ColDetectFieldEnabled=True; Kuka.CurrentCDSetIndex=0; Kuka.MovementParameterFieldEnabled=True; IlfCommand=SLIN
          ;ENDFOLD
          SLIN XP601 WITH $VEL = SVEL_CP(0.1, , LCPDAT27), $TOOL = STOOL2(FP601), $BASE = SBASE(FP601.BASE_NO), $IPO_MODE = SIPO_MODE(FP601.IPO_FRAME), $LOAD = SLOAD(FP601.TOOL_NO), $ACC = SACC_CP(LCPDAT27), $ORI_TYPE = SORI_TYP(LCPDAT27), $APO = SAPO(LCPDAT27), $JERK = SJERK(LCPDAT27), $COLLMON_TOL_PRO[1] = USE_CM_PRO_VALUES(0)
          ;ENDFOLD
          ;FOLD SLIN P602 Vel=0.1 m/s CPDAT27 Tool[1]:SMC Base[0] ;%{PE}
          ;FOLD Parameters ;%{h}
          ;Params IlfProvider=kukaroboter.basistech.inlineforms.movement.spline; Kuka.IsGlobalPoint=False; Kuka.PointName=P602; Kuka.BlendingEnabled=False; Kuka.MoveDataName=CPDAT27; Kuka.VelocityPath=0.1; Kuka.VelocityFieldEnabled=True; Kuka.ColDetectFieldEnabled=True; Kuka.CurrentCDSetIndex=0; Kuka.MovementParameterFieldEnabled=True; IlfCommand=SLIN
          ;ENDFOLD
          SLIN XP602 WITH $VEL = SVEL_CP(0.1, , LCPDAT27), $TOOL = STOOL2(FP602), $BASE = SBASE(FP602.BASE_NO), $IPO_MODE = SIPO_MODE(FP602.IPO_FRAME), $LOAD = SLOAD(FP602.TOOL_NO), $ACC = SACC_CP(LCPDAT27), $ORI_TYPE = SORI_TYP(LCPDAT27), $APO = SAPO(LCPDAT27), $JERK = SJERK(LCPDAT27), $COLLMON_TOL_PRO[1] = USE_CM_PRO_VALUES(0)
          ;ENDFOLD
        ENDIF

        IF finalPosition == 31 THEN
          ;FOLD SPTP P131 Vel=100 % PDAT1 Tool[1]:SMC Base[0] ;%{PE}
          ;FOLD Parameters ;%{h}
          ;Params IlfProvider=kukaroboter.basistech.inlineforms.movement.spline; Kuka.IsGlobalPoint=False; Kuka.PointName=P131; Kuka.BlendingEnabled=False; Kuka.MoveDataPtpName=PDAT1; Kuka.VelocityPtp=100; Kuka.VelocityFieldEnabled=True; Kuka.ColDetectFieldEnabled=True; Kuka.CurrentCDSetIndex=0; Kuka.MovementParameterFieldEnabled=True; IlfCommand=SPTP
          ;ENDFOLD
          SPTP XP131 WITH $VEL_AXIS[1] = SVEL_JOINT(100.0), $TOOL = STOOL2(FP131), $BASE = SBASE(FP131.BASE_NO), $IPO_MODE = SIPO_MODE(FP131.IPO_FRAME), $LOAD = SLOAD(FP131.TOOL_NO), $ACC_AXIS[1] = SACC_JOINT(PPDAT1), $APO = SAPO_PTP(PPDAT1), $GEAR_JERK[1] = SGEAR_JERK(PPDAT1), $COLLMON_TOL_PRO[1] = USE_CM_PRO_VALUES(0)
          ;ENDFOLD
          ;FOLD SLIN P231 Vel=0.1 m/s CPDAT27 Tool[1]:SMC Base[0] ;%{PE}
          ;FOLD Parameters ;%{h}
          ;Params IlfProvider=kukaroboter.basistech.inlineforms.movement.spline; Kuka.IsGlobalPoint=False; Kuka.PointName=P231; Kuka.BlendingEnabled=False; Kuka.MoveDataName=CPDAT27; Kuka.VelocityPath=0.1; Kuka.VelocityFieldEnabled=True; Kuka.ColDetectFieldEnabled=True; Kuka.CurrentCDSetIndex=0; Kuka.MovementParameterFieldEnabled=True; IlfCommand=SLIN
          ;ENDFOLD
          SLIN XP231 WITH $VEL = SVEL_CP(0.1, , LCPDAT27), $TOOL = STOOL2(FP231), $BASE = SBASE(FP231.BASE_NO), $IPO_MODE = SIPO_MODE(FP231.IPO_FRAME), $LOAD = SLOAD(FP231.TOOL_NO), $ACC = SACC_CP(LCPDAT27), $ORI_TYPE = SORI_TYP(LCPDAT27), $APO = SAPO(LCPDAT27), $JERK = SJERK(LCPDAT27), $COLLMON_TOL_PRO[1] = USE_CM_PRO_VALUES(0)
          ;ENDFOLD
          ;FOLD Gripper SET [1]Gripper1 State=[1]ABIERTA Wait 0.2[s] Check with Strategy 1 ;%{PE}
          ;FOLD Parameters Parameters ;%{h}
          ;Params IlfProvider=GripperTech.GripperSet;setgripper=1;setstate=1;setcont=nocont;waittime=0.2;errorstrategy=1
          ;ENDFOLD
          GRPg_SetStateAndCheck(1, 1, 0.2, 1)
          ;ENDFOLD
          ;FOLD SLIN P131 Vel=0.1 m/s CPDAT28 Tool[1]:SMC Base[0] ;%{PE}
          ;FOLD Parameters ;%{h}
          ;Params IlfProvider=kukaroboter.basistech.inlineforms.movement.spline; Kuka.IsGlobalPoint=False; Kuka.PointName=P131; Kuka.BlendingEnabled=False; Kuka.MoveDataName=CPDAT28; Kuka.VelocityPath=0.1; Kuka.VelocityFieldEnabled=True; Kuka.ColDetectFieldEnabled=True; Kuka.CurrentCDSetIndex=0; Kuka.MovementParameterFieldEnabled=True; IlfCommand=SLIN
          ;ENDFOLD
          SLIN XP131 WITH $VEL = SVEL_CP(0.1, , LCPDAT28), $TOOL = STOOL2(FP131), $BASE = SBASE(FP131.BASE_NO), $IPO_MODE = SIPO_MODE(FP131.IPO_FRAME), $LOAD = SLOAD(FP131.TOOL_NO), $ACC = SACC_CP(LCPDAT28), $ORI_TYPE = SORI_TYP(LCPDAT28), $APO = SAPO(LCPDAT28), $JERK = SJERK(LCPDAT28), $COLLMON_TOL_PRO[1] = USE_CM_PRO_VALUES(0)
          ;ENDFOLD
          ;FOLD SPTP P600 Vel=100 % PDAT1 Tool[1]:SMC Base[0] ;%{PE}
          ;FOLD Parameters ;%{h}
          ;Params IlfProvider=kukaroboter.basistech.inlineforms.movement.spline; Kuka.IsGlobalPoint=False; Kuka.PointName=P600; Kuka.BlendingEnabled=False; Kuka.MoveDataPtpName=PDAT1; Kuka.VelocityPtp=100; Kuka.VelocityFieldEnabled=True; Kuka.ColDetectFieldEnabled=True; Kuka.CurrentCDSetIndex=0; Kuka.MovementParameterFieldEnabled=True; IlfCommand=SPTP
          ;ENDFOLD
          SPTP XP600 WITH $VEL_AXIS[1] = SVEL_JOINT(100.0), $TOOL = STOOL2(FP600), $BASE = SBASE(FP600.BASE_NO), $IPO_MODE = SIPO_MODE(FP600.IPO_FRAME), $LOAD = SLOAD(FP600.TOOL_NO), $ACC_AXIS[1] = SACC_JOINT(PPDAT1), $APO = SAPO_PTP(PPDAT1), $GEAR_JERK[1] = SGEAR_JERK(PPDAT1), $COLLMON_TOL_PRO[1] = USE_CM_PRO_VALUES(0)
          ;ENDFOLD
          ;FOLD SLIN P601 Vel=0.1 m/s CPDAT27 Tool[1]:SMC Base[0] ;%{PE}
          ;FOLD Parameters ;%{h}
          ;Params IlfProvider=kukaroboter.basistech.inlineforms.movement.spline; Kuka.IsGlobalPoint=False; Kuka.PointName=P601; Kuka.BlendingEnabled=False; Kuka.MoveDataName=CPDAT27; Kuka.VelocityPath=0.1; Kuka.VelocityFieldEnabled=True; Kuka.ColDetectFieldEnabled=True; Kuka.CurrentCDSetIndex=0; Kuka.MovementParameterFieldEnabled=True; IlfCommand=SLIN
          ;ENDFOLD
          SLIN XP601 WITH $VEL = SVEL_CP(0.1, , LCPDAT27), $TOOL = STOOL2(FP601), $BASE = SBASE(FP601.BASE_NO), $IPO_MODE = SIPO_MODE(FP601.IPO_FRAME), $LOAD = SLOAD(FP601.TOOL_NO), $ACC = SACC_CP(LCPDAT27), $ORI_TYPE = SORI_TYP(LCPDAT27), $APO = SAPO(LCPDAT27), $JERK = SJERK(LCPDAT27), $COLLMON_TOL_PRO[1] = USE_CM_PRO_VALUES(0)
          ;ENDFOLD
          ;FOLD SLIN P602 Vel=0.1 m/s CPDAT27 Tool[1]:SMC Base[0] ;%{PE}
          ;FOLD Parameters ;%{h}
          ;Params IlfProvider=kukaroboter.basistech.inlineforms.movement.spline; Kuka.IsGlobalPoint=False; Kuka.PointName=P602; Kuka.BlendingEnabled=False; Kuka.MoveDataName=CPDAT27; Kuka.VelocityPath=0.1; Kuka.VelocityFieldEnabled=True; Kuka.ColDetectFieldEnabled=True; Kuka.CurrentCDSetIndex=0; Kuka.MovementParameterFieldEnabled=True; IlfCommand=SLIN
          ;ENDFOLD
          SLIN XP602 WITH $VEL = SVEL_CP(0.1, , LCPDAT27), $TOOL = STOOL2(FP602), $BASE = SBASE(FP602.BASE_NO), $IPO_MODE = SIPO_MODE(FP602.IPO_FRAME), $LOAD = SLOAD(FP602.TOOL_NO), $ACC = SACC_CP(LCPDAT27), $ORI_TYPE = SORI_TYP(LCPDAT27), $APO = SAPO(LCPDAT27), $JERK = SJERK(LCPDAT27), $COLLMON_TOL_PRO[1] = USE_CM_PRO_VALUES(0)
          ;ENDFOLD
        ENDIF

